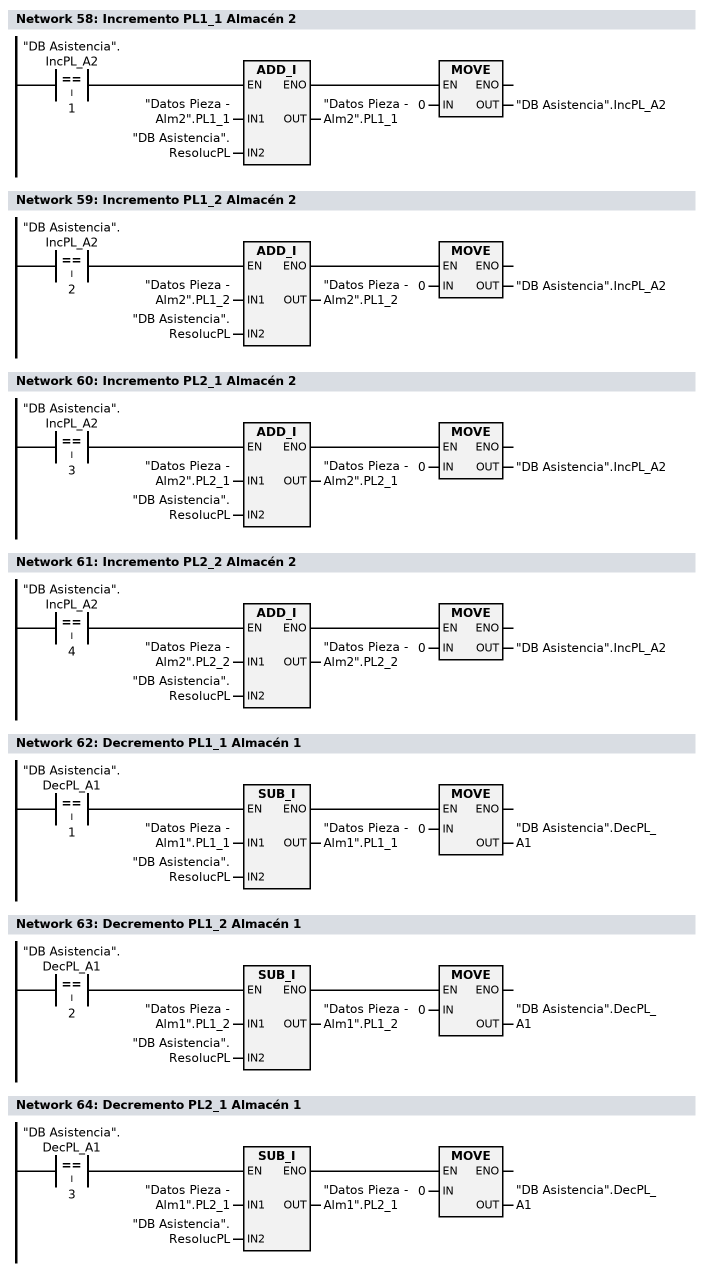
NETWORK
TITLE = Incremento PL1_1 Almacén 2
      A(;
      A(;
      L     "DB Asistencia".IncPL_A2;
      L     1;
      ==I;
      );
      JNB   _03d;
      L     "Datos Pieza - Alm2".PL1_1;
      L     "DB Asistencia".ResolucPL;
      +I;
      T     "Datos Pieza - Alm2".PL1_1;
      AN    OV;
      SAVE;
      CLR;
_03d: A     BR;
      );
      JNB   _03e;
      L     0;
      T     "DB Asistencia".IncPL_A2;
_03e: NOP   0;
NETWORK
TITLE = Incremento PL1_2 Almacén 2
      A(;
      A(;
      L     "DB Asistencia".IncPL_A2;
      L     2;
      ==I;
      );
      JNB   _03f;
      L     "Datos Pieza - Alm2".PL1_2;
      L     "DB Asistencia".ResolucPL;
      +I;
      T     "Datos Pieza - Alm2".PL1_2;
      AN    OV;
      SAVE;
      CLR;
_03f: A     BR;
      );
      JNB   _040;
      L     0;
      T     "DB Asistencia".IncPL_A2;
_040: NOP   0;
NETWORK
TITLE = Incremento PL2_1 Almacén 2
      A(;
      A(;
      L     "DB Asistencia".IncPL_A2;
      L     3;
      ==I;
      );
      JNB   _041;
      L     "Datos Pieza - Alm2".PL2_1;
      L     "DB Asistencia".ResolucPL;
      +I;
      T     "Datos Pieza - Alm2".PL2_1;
      AN    OV;
      SAVE;
      CLR;
_041: A     BR;
      );
      JNB   _042;
      L     0;
      T     "DB Asistencia".IncPL_A2;
_042: NOP   0;
NETWORK
TITLE = Incremento PL2_2 Almacén 2
      A(;
      A(;
      L     "DB Asistencia".IncPL_A2;
      L     4;
      ==I;
      );
      JNB   _043;
      L     "Datos Pieza - Alm2".PL2_2;
      L     "DB Asistencia".ResolucPL;
      +I;
      T     "Datos Pieza - Alm2".PL2_2;
      AN    OV;
      SAVE;
      CLR;
_043: A     BR;
      );
      JNB   _044;
      L     0;
      T     "DB Asistencia".IncPL_A2;
_044: NOP   0;
NETWORK
TITLE = Decremento PL1_1 Almacén 1
      A(;
      A(;
      L     "DB Asistencia".DecPL_A1;
      L     1;
      ==I;
      );
      JNB   _045;
      L     "Datos Pieza - Alm1".PL1_1;
      L     "DB Asistencia".ResolucPL;
      -I;
      T     "Datos Pieza - Alm1".PL1_1;
      AN    OV;
      SAVE;
      CLR;
_045: A     BR;
      );
      JNB   _046;
      L     0;
      T     "DB Asistencia".DecPL_A1;
_046: NOP   0;
NETWORK
TITLE = Decremento PL1_2 Almacén 1
      A(;
      A(;
      L     "DB Asistencia".DecPL_A1;
      L     2;
      ==I;
      );
      JNB   _047;
      L     "Datos Pieza - Alm1".PL1_2;
      L     "DB Asistencia".ResolucPL;
      -I;
      T     "Datos Pieza - Alm1".PL1_2;
      AN    OV;
      SAVE;
      CLR;
_047: A     BR;
      );
      JNB   _048;
      L     0;
      T     "DB Asistencia".DecPL_A1;
_048: NOP   0;
NETWORK
TITLE = Decremento PL2_1 Almacén 1
      A(;
      A(;
      L     "DB Asistencia".DecPL_A1;
      L     3;
      ==I;
      );
      JNB   _049;
      L     "Datos Pieza - Alm1".PL2_1;
      L     "DB Asistencia".ResolucPL;
      -I;
      T     "Datos Pieza - Alm1".PL2_1;
      AN    OV;
      SAVE;
      CLR;
_049: A     BR;
      );
      JNB   _04a;
      L     0;
      T     "DB Asistencia".DecPL_A1;
_04a: NOP   0;
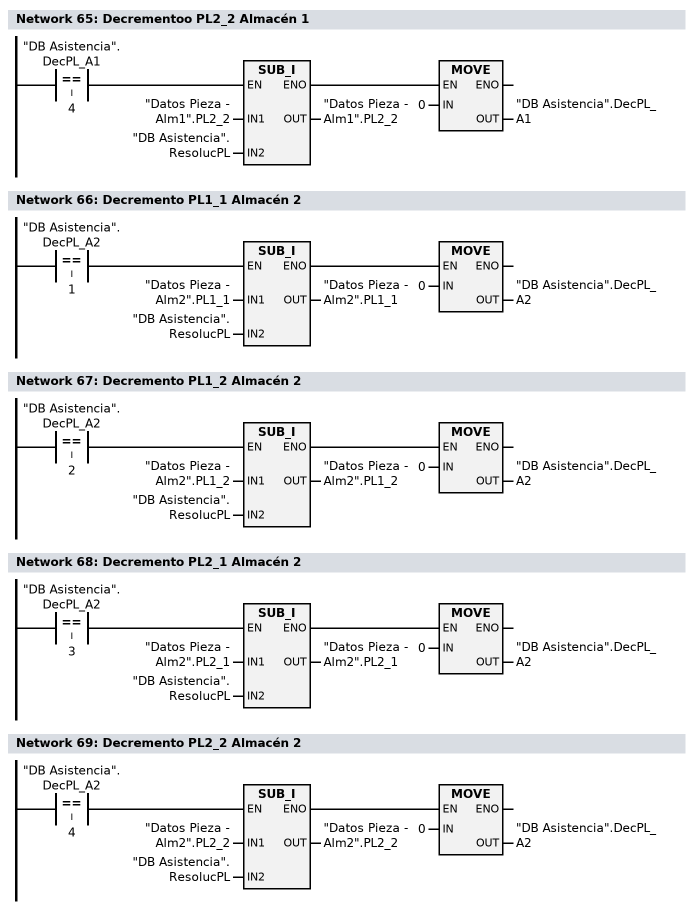
NETWORK
TITLE = Decrementoo PL2_2 Almacén 1
      A(;
      A(;
      L     "DB Asistencia".DecPL_A1;
      L     4;
      ==I;
      );
      JNB   _04b;
      L     "Datos Pieza - Alm1".PL2_2;
      L     "DB Asistencia".ResolucPL;
      -I;
      T     "Datos Pieza - Alm1".PL2_2;
      AN    OV;
      SAVE;
      CLR;
_04b: A     BR;
      );
      JNB   _04c;
      L     0;
      T     "DB Asistencia".DecPL_A1;
_04c: NOP   0;
NETWORK
TITLE = Decremento PL1_1 Almacén 2
      A(;
      A(;
      L     "DB Asistencia".DecPL_A2;
      L     1;
      ==I;
      );
      JNB   _04d;
      L     "Datos Pieza - Alm2".PL1_1;
      L     "DB Asistencia".ResolucPL;
      -I;
      T     "Datos Pieza - Alm2".PL1_1;
      AN    OV;
      SAVE;
      CLR;
_04d: A     BR;
      );
      JNB   _04e;
      L     0;
      T     "DB Asistencia".DecPL_A2;
_04e: NOP   0;
NETWORK
TITLE = Decremento PL1_2 Almacén 2
      A(;
      A(;
      L     "DB Asistencia".DecPL_A2;
      L     2;
      ==I;
      );
      JNB   _04f;
      L     "Datos Pieza - Alm2".PL1_2;
      L     "DB Asistencia".ResolucPL;
      -I;
      T     "Datos Pieza - Alm2".PL1_2;
      AN    OV;
      SAVE;
      CLR;
_04f: A     BR;
      );
      JNB   _050;
      L     0;
      T     "DB Asistencia".DecPL_A2;
_050: NOP   0;
NETWORK
TITLE = Decremento PL2_1 Almacén 2
      A(;
      A(;
      L     "DB Asistencia".DecPL_A2;
      L     3;
      ==I;
      );
      JNB   _051;
      L     "Datos Pieza - Alm2".PL2_1;
      L     "DB Asistencia".ResolucPL;
      -I;
      T     "Datos Pieza - Alm2".PL2_1;
      AN    OV;
      SAVE;
      CLR;
_051: A     BR;
      );
      JNB   _052;
      L     0;
      T     "DB Asistencia".DecPL_A2;
_052: NOP   0;
NETWORK
TITLE = Decremento PL2_2 Almacén 2
      A(;
      A(;
      L     "DB Asistencia".DecPL_A2;
      L     4;
      ==I;
      );
      JNB   _053;
      L     "Datos Pieza - Alm2".PL2_2;
      L     "DB Asistencia".ResolucPL;
      -I;
      T     "Datos Pieza - Alm2".PL2_2;
      AN    OV;
      SAVE;
      CLR;
_053: A     BR;
      );
      JNB   _054;
      L     0;
      T     "DB Asistencia".DecPL_A2;
_054: NOP   0;
END_FUNCTION

FUNCTION "Control de Plegadora" : VOID	// FC 9
TITLE = Control de Plegadora
AUTHOR : EMR
NAME : eProC
VERSION : 0.1
VAR_TEMP
  AUX_POS_RECEPCION : DINT ;
  AUX_POS_ALINEACION : DINT ;
  AUX_POS_PL1 : DINT ;
  AUX_POS_PL2 : DINT ;
  AUX_POS_ENTREGA : DINT ;
  AUX_SALIDA : DINT ;
  AUX_CHAPA_COMPLETA : DINT ;
  AUX_ESPERA : DINT ;
  PL1_A : DINT ;
  PL1_B : DINT ;
  PL1_C : DINT ;
  PL1_D : DINT ;
  PL1_1 : DINT ;
  PL1_2 : DINT ;
  AUX_ENCODER : REAL ;
  AUX_ENCODER2 : DINT ;
  AUX_REAL : REAL ;
  AUX_REAL2 : REAL ;
  AUX_REAL3 : REAL ;
  PL2_1 : DINT ;
  PL2_2 : DINT ;
  POS_PINZA_SEGURA1 : DINT ;
  POS_PINZA_SEGURA2 : DINT ;
  AUX_DINT : DINT ;
  AUX_POS_RECEP : BOOL ;	//Plegadores en Posición Recepción
  AUX_POS_ALIN : BOOL ;	//Plegadores en Posición Alineación
  AUX_POS_ENT : BOOL ;	//Plegadores en Posición Entrega
  AUX_POS_ESP : BOOL ;	//Plegadores en Posición Espera
  AUX_POS_26 : BOOL ;
  AUX_POS_25 : BOOL ;
  AUX_POS_PLEG2 : BOOL ;	//Plegadores en Posición Plegado 2
  AUX_POS_24 : BOOL ;
  AUX_POS_22 : BOOL ;
  AUX_POS_PLEG1 : BOOL ;	//Plegadores en Posición Plegado 1
  AUX_POS_23 : BOOL ;
  AUX_POS_21 : BOOL ;
END_VAR
BEGIN
NETWORK
TITLE = ------------- HABILITACIÓN SERVOS -----------------
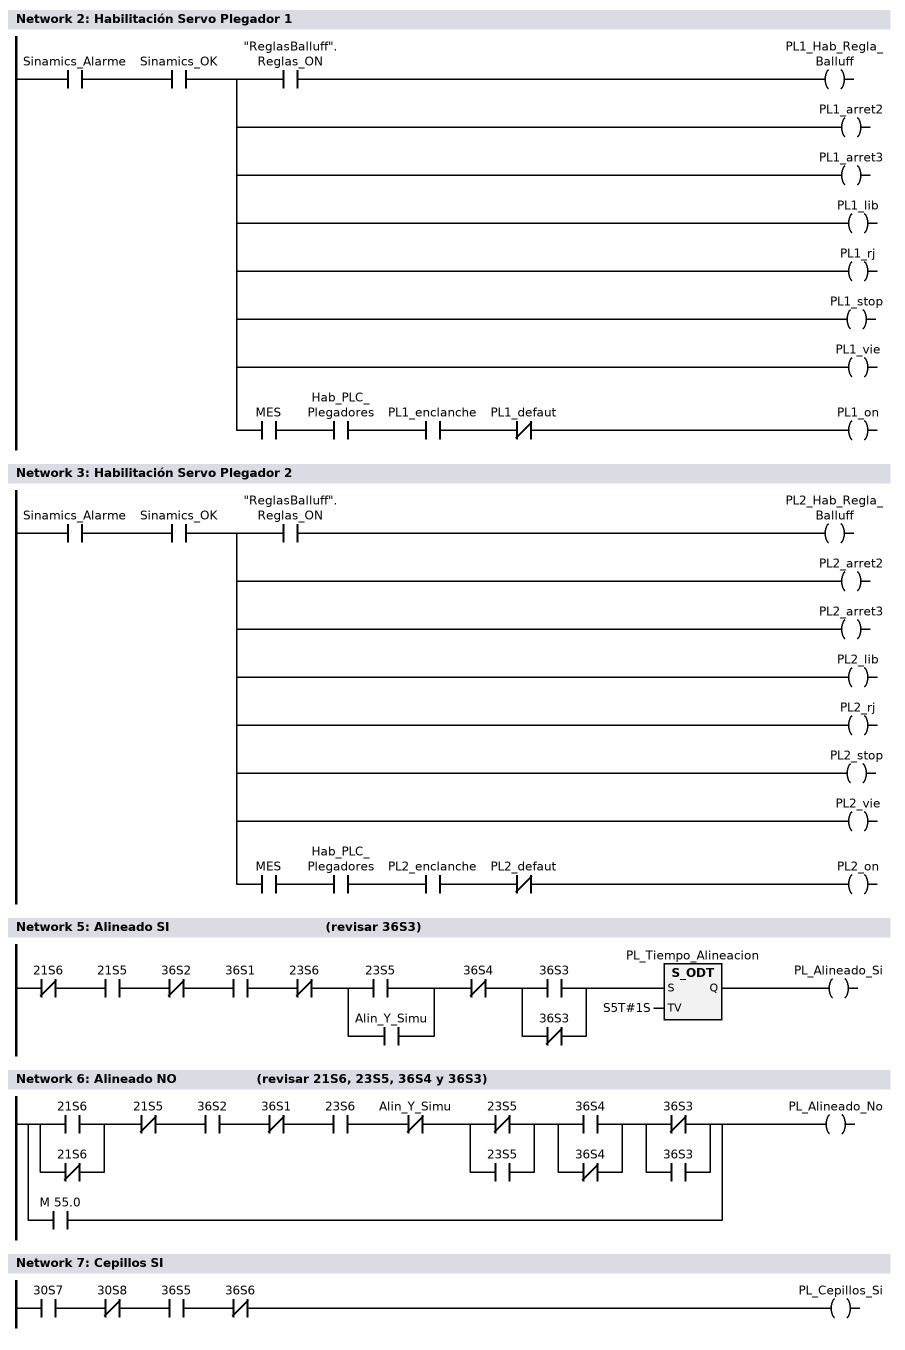
NETWORK
TITLE = Habilitación Servo Plegador 1
      A     "Sinamics_Alarme";
      A     "Sinamics_OK";
      =     L 98.0;
      A     L 98.0;
      A     "ReglasBalluff".Reglas_ON;
      =     "PL1_Hab_Regla_Balluff";
      A     L 98.0;
      BLD   102;
      =     "PL1_arret2";
      A     L 98.0;
      BLD   102;
      =     "PL1_arret3";
      A     L 98.0;
      BLD   102;
      =     "PL1_lib";
      A     L 98.0;
      BLD   102;
      =     "PL1_rj";
      A     L 98.0;
      BLD   102;
      =     "PL1_stop";
      A     L 98.0;
      BLD   102;
      =     "PL1_vie";
      A     L 98.0;
      A     "MES";
      A     "Hab_PLC_Plegadores";
      A     "PL1_enclanche";
      AN    "PL1_defaut";
      =     "PL1_on";
NETWORK
TITLE = Habilitación Servo Plegador 2
      A     "Sinamics_Alarme";
      A     "Sinamics_OK";
      =     L 98.0;
      A     L 98.0;
      A     "ReglasBalluff".Reglas_ON;
      =     "PL2_Hab_Regla_Balluff";
      A     L 98.0;
      BLD   102;
      =     "PL2_arret2";
      A     L 98.0;
      BLD   102;
      =     "PL2_arret3";
      A     L 98.0;
      BLD   102;
      =     "PL2_lib";
      A     L 98.0;
      BLD   102;
      =     "PL2_rj";
      A     L 98.0;
      BLD   102;
      =     "PL2_stop";
      A     L 98.0;
      BLD   102;
      =     "PL2_vie";
      A     L 98.0;
      A     "MES";
      A     "Hab_PLC_Plegadores";
      A     "PL2_enclanche";
      AN    "PL2_defaut";
      =     "PL2_on";
NETWORK
TITLE = ------------- RESUMEN DE SENSORES -----------------
NETWORK
TITLE = Alineado SI                                       (revisar 36S3)
      AN    "21S6";
      A     "21S5";
      AN    "36S2";
      A     "36S1";
      AN    "23S6";
      A(;
      O     "23S5";
      O     "Alin_Y_Simu";
      );
      AN    "36S4";
      A(;
      O     "36S3";
      ON    "36S3";
      );
      L     S5T#1S;
      SD    "PL_Tiempo_Alineacion";
      NOP   0;
      NOP   0;
      NOP   0;
      A     "PL_Tiempo_Alineacion";
      =     "PL_Alineado_Si";
NETWORK
TITLE = Alineado NO                    (revisar 21S6, 23S5, 36S4 y 36S3)
      A(;
      O     "21S6";
      ON    "21S6";
      );
      AN    "21S5";
      A     "36S2";
      AN    "36S1";
      A     "23S6";
      AN    "Alin_Y_Simu";
      A(;
      ON    "23S5";
      O     "23S5";
      );
      A(;
      O     "36S4";
      ON    "36S4";
      );
      A(;
      ON    "36S3";
      O     "36S3";
      );
      O     M 55.0;
      =     "PL_Alineado_No";
NETWORK
TITLE = Cepillos SI
      A     "30S7";
      AN    "30S8";
      A     "36S5";
      AN    "36S6";
      =     "PL_Cepillos_Si";
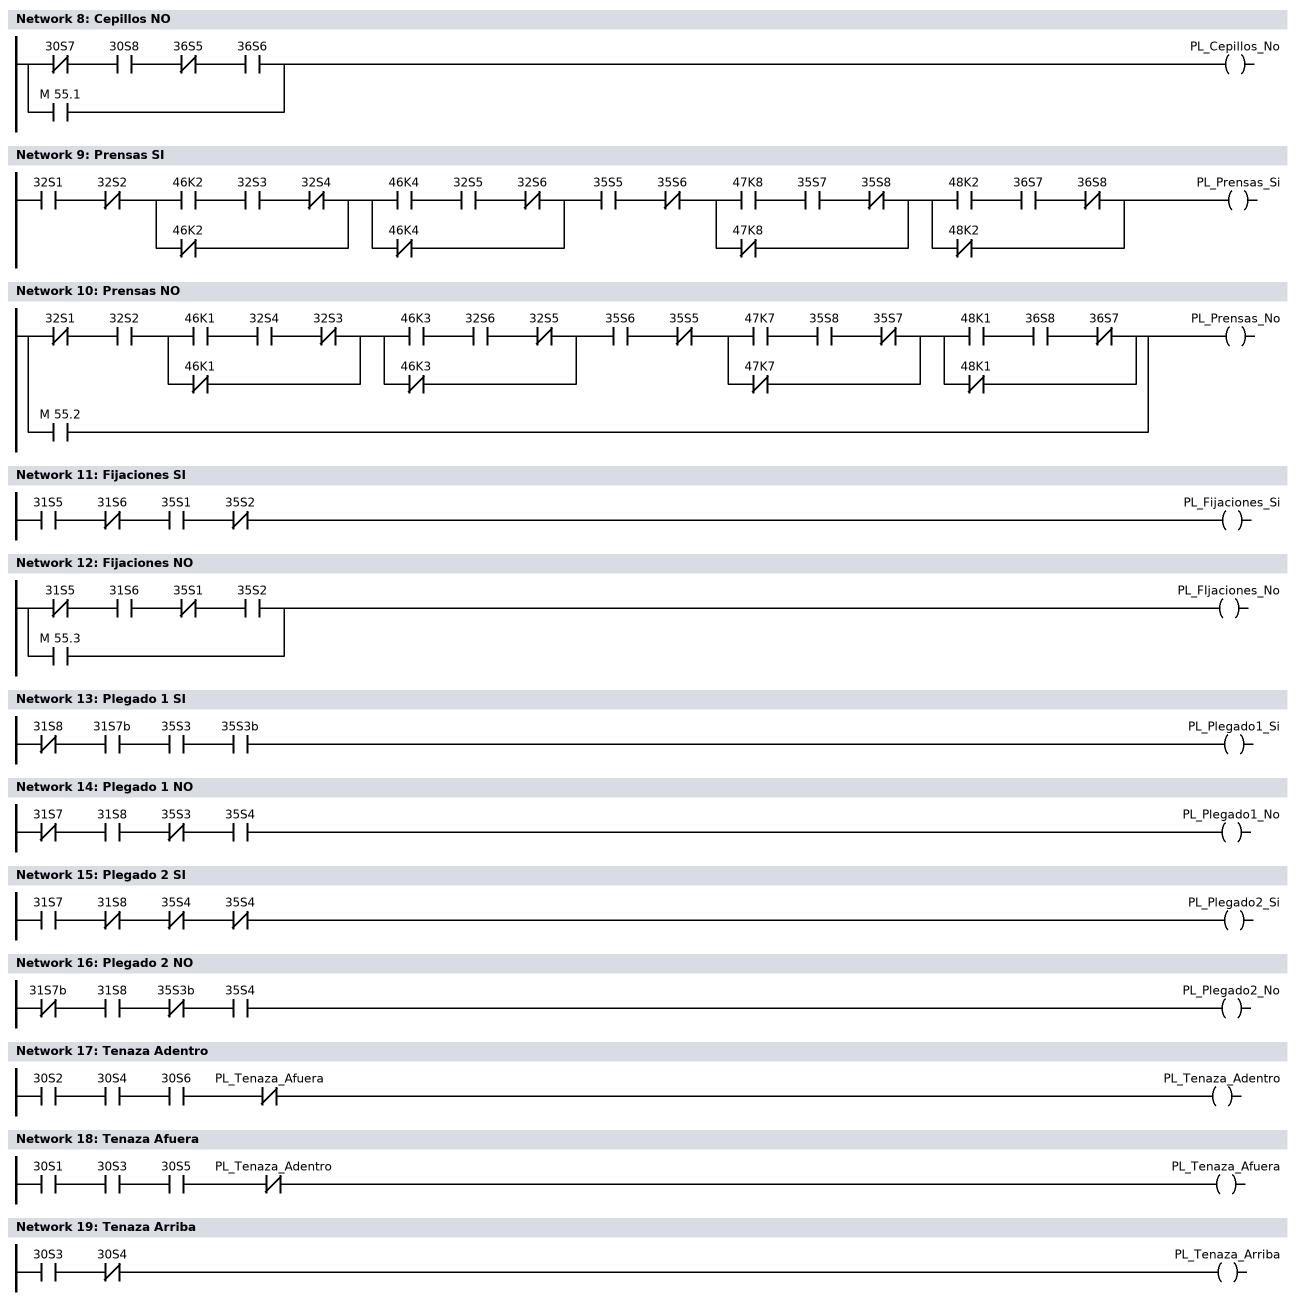
NETWORK
TITLE = Cepillos NO
      AN    "30S7";
      A     "30S8";
      AN    "36S5";
      A     "36S6";
      O     M 55.1;
      =     "PL_Cepillos_No";
NETWORK
TITLE = Prensas SI
      A     "32S1";
      AN    "32S2";
      A(;
      A     "46K2";
      A     "32S3";
      AN    "32S4";
      ON    "46K2";
      );
      A(;
      A     "46K4";
      A     "32S5";
      AN    "32S6";
      ON    "46K4";
      );
      A     "35S5";
      AN    "35S6";
      A(;
      A     "47K8";
      A     "35S7";
      AN    "35S8";
      ON    "47K8";
      );
      A(;
      A     "48K2";
      A     "36S7";
      AN    "36S8";
      ON    "48K2";
      );
      =     "PL_Prensas_Si";
NETWORK
TITLE = Prensas NO
      AN    "32S1";
      A     "32S2";
      A(;
      A     "46K1";
      A     "32S4";
      AN    "32S3";
      ON    "46K1";
      );
      A(;
      A     "46K3";
      A     "32S6";
      AN    "32S5";
      ON    "46K3";
      );
      A     "35S6";
      AN    "35S5";
      A(;
      A     "47K7";
      A     "35S8";
      AN    "35S7";
      ON    "47K7";
      );
      A(;
      A     "48K1";
      A     "36S8";
      AN    "36S7";
      ON    "48K1";
      );
      O     M 55.2;
      =     "PL_Prensas_No";
NETWORK
TITLE = Fijaciones SI
      A     "31S5";
      AN    "31S6";
      A     "35S1";
      AN    "35S2";
      =     "PL_Fijaciones_Si";
NETWORK
TITLE = Fijaciones NO
      AN    "31S5";
      A     "31S6";
      AN    "35S1";
      A     "35S2";
      O     M 55.3;
      =     "PL_FIjaciones_No";
NETWORK
TITLE = Plegado 1 SI
      AN    "31S8";
      A     "31S7b";
      A     "35S3";
      A     "35S3b";
      =     "PL_Plegado1_Si";
NETWORK
TITLE = Plegado 1 NO
      AN    "31S7";
      A     "31S8";
      AN    "35S3";
      A     "35S4";
      =     "PL_Plegado1_No";
NETWORK
TITLE = Plegado 2 SI
      A     "31S7";
      AN    "31S8";
      AN    "35S4";
      AN    "35S4";
      =     "PL_Plegado2_Si";
NETWORK
TITLE = Plegado 2 NO
      AN    "31S7b";
      A     "31S8";
      AN    "35S3b";
      A     "35S4";
      =     "PL_Plegado2_No";
NETWORK
TITLE = Tenaza Adentro
      A     "30S2";
      A     "30S4";
      A     "30S6";
      AN    "PL_Tenaza_Afuera";
      =     "PL_Tenaza_Adentro";
NETWORK
TITLE = Tenaza Afuera
      A     "30S1";
      A     "30S3";
      A     "30S5";
      AN    "PL_Tenaza_Adentro";
      =     "PL_Tenaza_Afuera";
NETWORK
TITLE = Tenaza Arriba
      A     "30S3";
      AN    "30S4";
      =     "PL_Tenaza_Arriba";
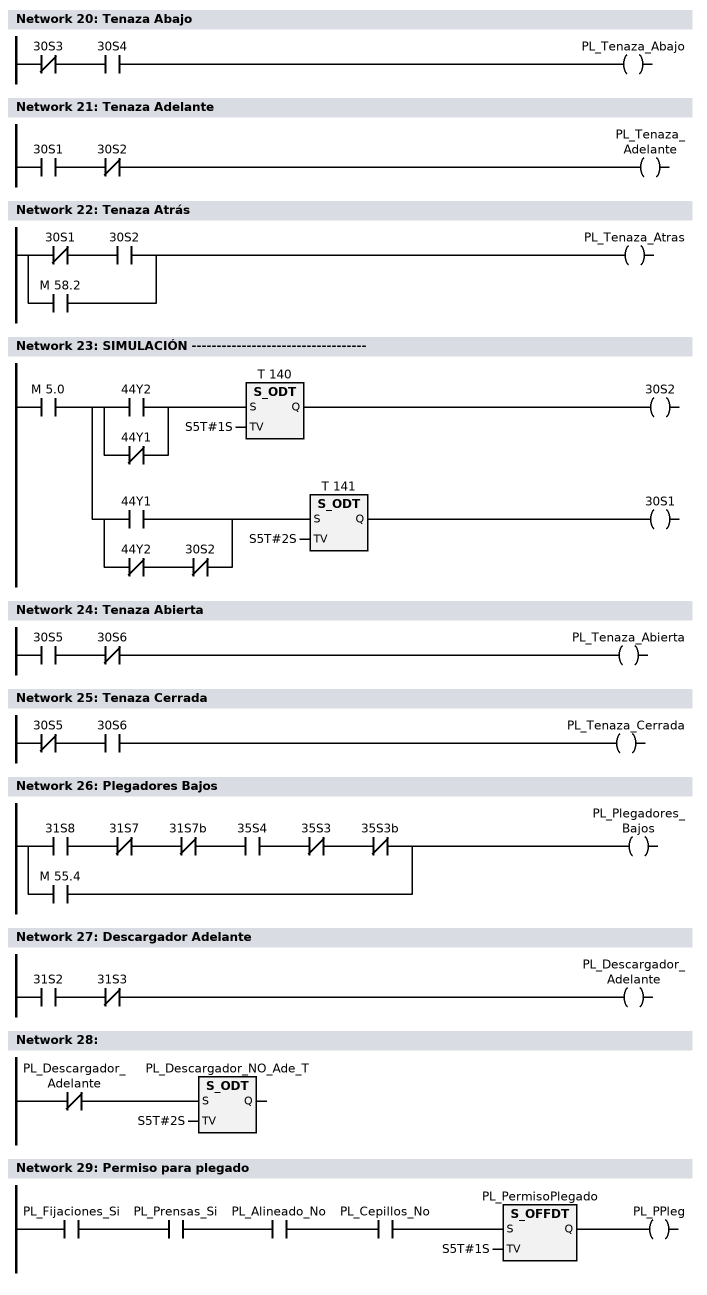
NETWORK
TITLE = Tenaza Abajo
      AN    "30S3";
      A     "30S4";
      =     "PL_Tenaza_Abajo";
NETWORK
TITLE = Tenaza Adelante
      A     "30S1";
      AN    "30S2";
      =     "PL_Tenaza_Adelante";
NETWORK
TITLE = Tenaza Atrás
      AN    "30S1";
      A     "30S2";
      O     M 58.2;
      =     "PL_Tenaza_Atras";
NETWORK
TITLE = SIMULACIÓN -----------------------------------
      A     M 5.0;
      =     L 98.0;
      A     L 98.0;
      A(;
      O     "44Y2";
      ON    "44Y1";
      );
      L     S5T#1S;
      SD    T 140;
      NOP   0;
      NOP   0;
      NOP   0;
      A     T 140;
      =     "30S2";
      A     L 98.0;
      A(;
      O     "44Y1";
      O;
      AN    "44Y2";
      AN    "30S2";
      );
      L     S5T#2S;
      SD    T 141;
      NOP   0;
      NOP   0;
      NOP   0;
      A     T 141;
      =     "30S1";
NETWORK
TITLE = Tenaza Abierta
      A     "30S5";
      AN    "30S6";
      =     "PL_Tenaza_Abierta";
NETWORK
TITLE = Tenaza Cerrada
      AN    "30S5";
      A     "30S6";
      =     "PL_Tenaza_Cerrada";
NETWORK
TITLE = Plegadores Bajos
      A     "31S8";
      AN    "31S7";
      AN    "31S7b";
      A     "35S4";
      AN    "35S3";
      AN    "35S3b";
      O     M 55.4;
      =     "PL_Plegadores_Bajos";
NETWORK
TITLE = Descargador Adelante
      A     "31S2";
      AN    "31S3";
      =     "PL_Descargador_Adelante";
NETWORK
TITLE =
      AN    "PL_Descargador_Adelante";
      L     S5T#2S;
      SD    "PL_Descargador_NO_Ade_T";
      NOP   0;
      NOP   0;
      NOP   0;
      NOP   0;
NETWORK
TITLE = Permiso para plegado
      A     "PL_Fijaciones_Si";
      A     "PL_Prensas_Si";
      A     "PL_Alineado_No";
      A     "PL_Cepillos_No";
      L     S5T#1S;
      SF    "PL_PermisoPlegado";
      NOP   0;
      NOP   0;
      NOP   0;
      A     "PL_PermisoPlegado";
      =     "PL_PPleg";
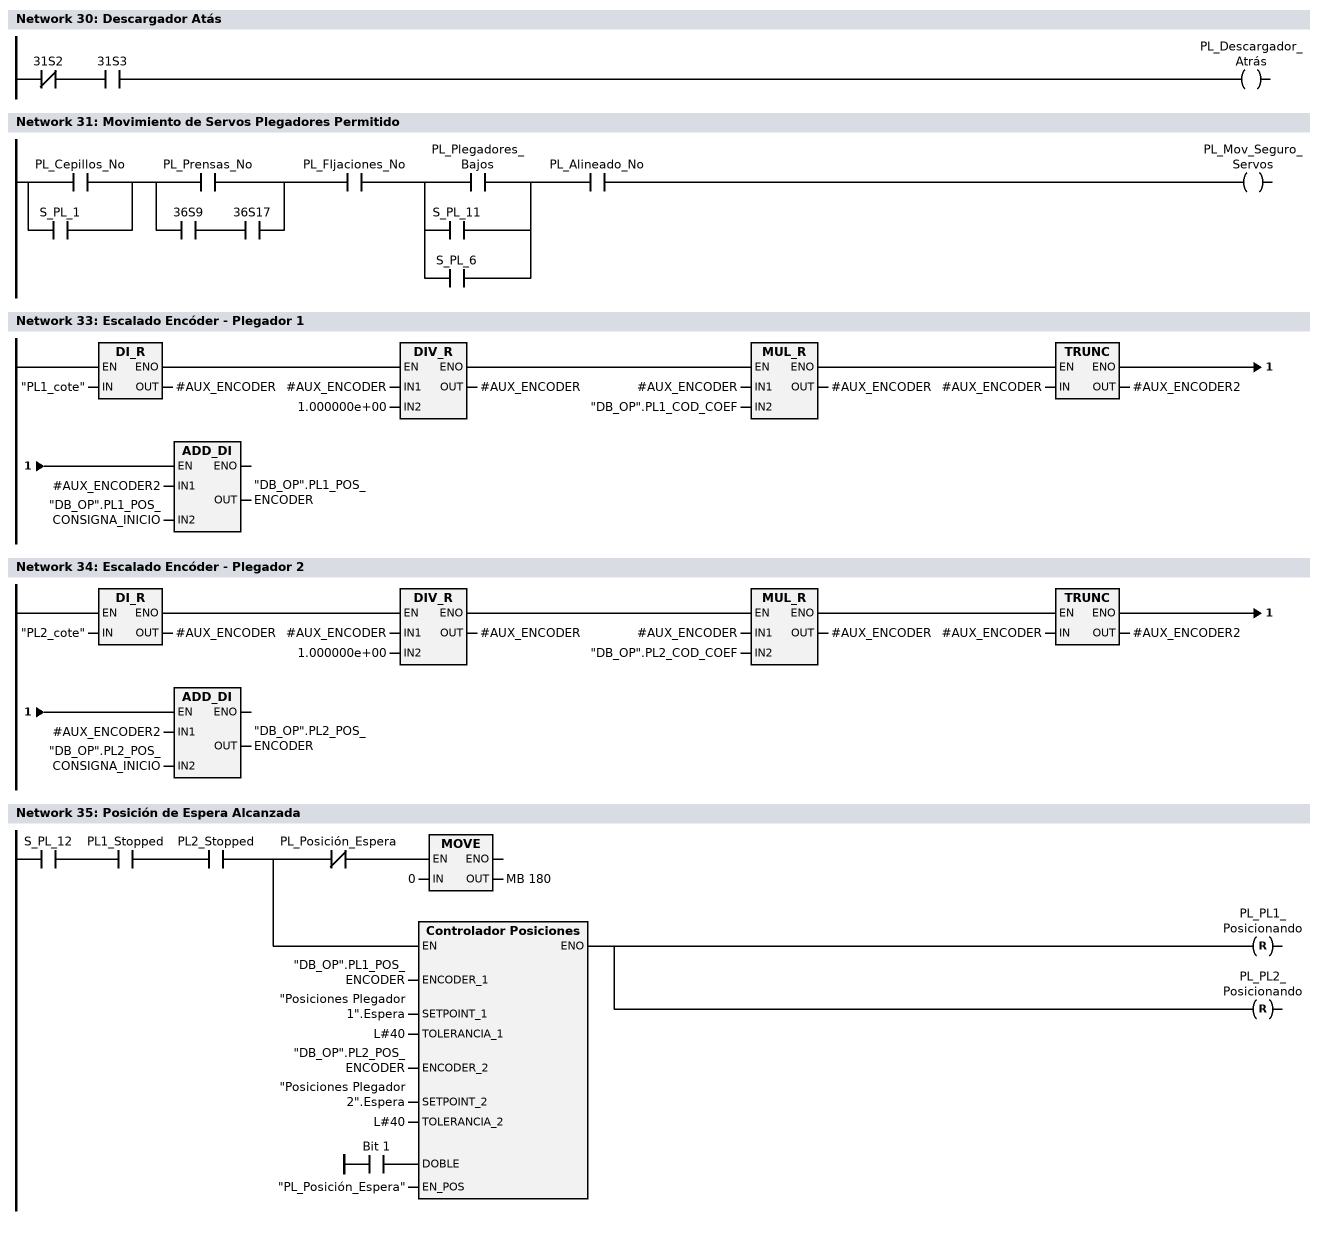
NETWORK
TITLE = Descargador Atás
      AN    "31S2";
      A     "31S3";
      =     "PL_Descargador_Atrás";
NETWORK
TITLE = Movimiento de Servos Plegadores Permitido
      A(;
      O     "PL_Cepillos_No";
      O     "S_PL_1";
      );
      A(;
      O     "PL_Prensas_No";
      O;
      A     "36S9";
      A     "36S17";
      );
      A     "PL_FIjaciones_No";
      A(;
      O     "PL_Plegadores_Bajos";
      O     "S_PL_11";
      O     "S_PL_6";
      );
      A     "PL_Alineado_No";
      =     "PL_Mov_Seguro_Servos";
NETWORK
TITLE = ------------ ESCALADO DE ENCODERS -------------
NETWORK
TITLE = Escalado Encóder - Plegador 1
      A(;
      A(;
      A(;
      A(;
      L     "PL1_cote";
      DTR;
      T     #AUX_ENCODER;
      SET;
      SAVE;
      CLR;
      A     BR;
      );
      JNB   _001;
      L     #AUX_ENCODER;
      L     1.000000e+00;
      /R;
      T     #AUX_ENCODER;
      AN    OV;
      SAVE;
      CLR;
_001: A     BR;
      );
      JNB   _002;
      L     #AUX_ENCODER;
      L     "DB_OP".PL1_COD_COEF;
      *R;
      T     #AUX_ENCODER;
      AN    OV;
      SAVE;
      CLR;
_002: A     BR;
      );
      JNB   _003;
      L     #AUX_ENCODER;
      TRUNC;
      T     #AUX_ENCODER2;
      AN    OV;
      SAVE;
      CLR;
_003: A     BR;
      );
      JNB   _004;
      L     #AUX_ENCODER2;
      L     "DB_OP".PL1_POS_CONSIGNA_INICIO;
      +D;
      T     "DB_OP".PL1_POS_ENCODER;
_004: NOP   0;
NETWORK
TITLE = Escalado Encóder - Plegador 2
      A(;
      A(;
      A(;
      A(;
      L     "PL2_cote";
      DTR;
      T     #AUX_ENCODER;
      SET;
      SAVE;
      CLR;
      A     BR;
      );
      JNB   _005;
      L     #AUX_ENCODER;
      L     1.000000e+00;
      /R;
      T     #AUX_ENCODER;
      AN    OV;
      SAVE;
      CLR;
_005: A     BR;
      );
      JNB   _006;
      L     #AUX_ENCODER;
      L     "DB_OP".PL2_COD_COEF;
      *R;
      T     #AUX_ENCODER;
      AN    OV;
      SAVE;
      CLR;
_006: A     BR;
      );
      JNB   _007;
      L     #AUX_ENCODER;
      TRUNC;
      T     #AUX_ENCODER2;
      AN    OV;
      SAVE;
      CLR;
_007: A     BR;
      );
      JNB   _008;
      L     #AUX_ENCODER2;
      L     "DB_OP".PL2_POS_CONSIGNA_INICIO;
      +D;
      T     "DB_OP".PL2_POS_ENCODER;
_008: NOP   0;
NETWORK
TITLE = Posición de Espera Alcanzada
      A     "S_PL_12";
      A     "PL1_Stopped";
      A     "PL2_Stopped";
      =     L 98.0;
      A     L 98.0;
      AN    "PL_Posición_Espera";
      JNB   _009;
      L     0;
      T     MB 180;
_009: NOP   0;
      A     "Bit 1";
      =     L 98.1;
      BLD   103;
      A     L 98.0;
      JNB   _00a;
      CALL  "Controlador Posiciones" (
           ENCODER_1                := "DB_OP".PL1_POS_ENCODER,
           SETPOINT_1               := "Posiciones Plegador 1".Espera,
           TOLERANCIA_1             := L#40,
           ENCODER_2                := "DB_OP".PL2_POS_ENCODER,
           SETPOINT_2               := "Posiciones Plegador 2".Espera,
           TOLERANCIA_2             := L#40,
           DOBLE                    := L 98.1,
           EN_POS                   := "PL_Posición_Espera");
_00a: A     BR;
      R     "PL_PL1_Posicionando";
      R     "PL_PL2_Posicionando";
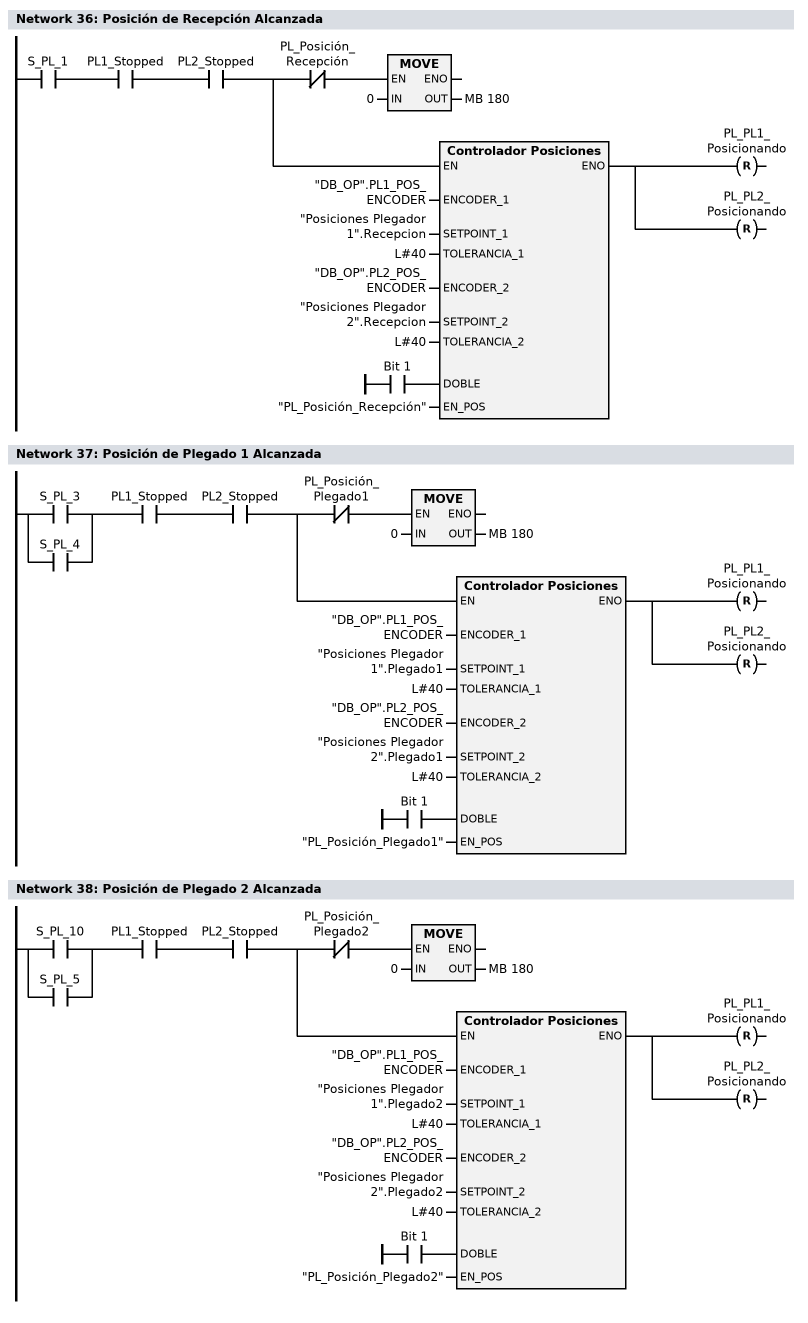
NETWORK
TITLE = Posición de Recepción Alcanzada
      A     "S_PL_1";
      A     "PL1_Stopped";
      A     "PL2_Stopped";
      =     L 98.0;
      A     L 98.0;
      AN    "PL_Posición_Recepción";
      JNB   _00b;
      L     0;
      T     MB 180;
_00b: NOP   0;
      A     "Bit 1";
      =     L 98.1;
      BLD   103;
      A     L 98.0;
      JNB   _00c;
      CALL  "Controlador Posiciones" (
           ENCODER_1                := "DB_OP".PL1_POS_ENCODER,
           SETPOINT_1               := "Posiciones Plegador 1".Recepcion,
           TOLERANCIA_1             := L#40,
           ENCODER_2                := "DB_OP".PL2_POS_ENCODER,
           SETPOINT_2               := "Posiciones Plegador 2".Recepcion,
           TOLERANCIA_2             := L#40,
           DOBLE                    := L 98.1,
           EN_POS                   := "PL_Posición_Recepción");
_00c: A     BR;
      R     "PL_PL1_Posicionando";
      R     "PL_PL2_Posicionando";
NETWORK
TITLE = Posición de Plegado 1 Alcanzada
      A(;
      O     "S_PL_3";
      O     "S_PL_4";
      );
      A     "PL1_Stopped";
      A     "PL2_Stopped";
      =     L 98.0;
      A     L 98.0;
      AN    "PL_Posición_Plegado1";
      JNB   _00d;
      L     0;
      T     MB 180;
_00d: NOP   0;
      A     "Bit 1";
      =     L 98.1;
      BLD   103;
      A     L 98.0;
      JNB   _00e;
      CALL  "Controlador Posiciones" (
           ENCODER_1                := "DB_OP".PL1_POS_ENCODER,
           SETPOINT_1               := "Posiciones Plegador 1".Plegado1,
           TOLERANCIA_1             := L#40,
           ENCODER_2                := "DB_OP".PL2_POS_ENCODER,
           SETPOINT_2               := "Posiciones Plegador 2".Plegado1,
           TOLERANCIA_2             := L#40,
           DOBLE                    := L 98.1,
           EN_POS                   := "PL_Posición_Plegado1");
_00e: A     BR;
      R     "PL_PL1_Posicionando";
      R     "PL_PL2_Posicionando";
NETWORK
TITLE = Posición de Plegado 2 Alcanzada
      A(;
      O     "S_PL_10";
      O     "S_PL_5";
      );
      A     "PL1_Stopped";
      A     "PL2_Stopped";
      =     L 98.0;
      A     L 98.0;
      AN    "PL_Posición_Plegado2";
      JNB   _00f;
      L     0;
      T     MB 180;
_00f: NOP   0;
      A     "Bit 1";
      =     L 98.1;
      BLD   103;
      A     L 98.0;
      JNB   _010;
      CALL  "Controlador Posiciones" (
           ENCODER_1                := "DB_OP".PL1_POS_ENCODER,
           SETPOINT_1               := "Posiciones Plegador 1".Plegado2,
           TOLERANCIA_1             := L#40,
           ENCODER_2                := "DB_OP".PL2_POS_ENCODER,
           SETPOINT_2               := "Posiciones Plegador 2".Plegado2,
           TOLERANCIA_2             := L#40,
           DOBLE                    := L 98.1,
           EN_POS                   := "PL_Posición_Plegado2");
_010: A     BR;
      R     "PL_PL1_Posicionando";
      R     "PL_PL2_Posicionando";
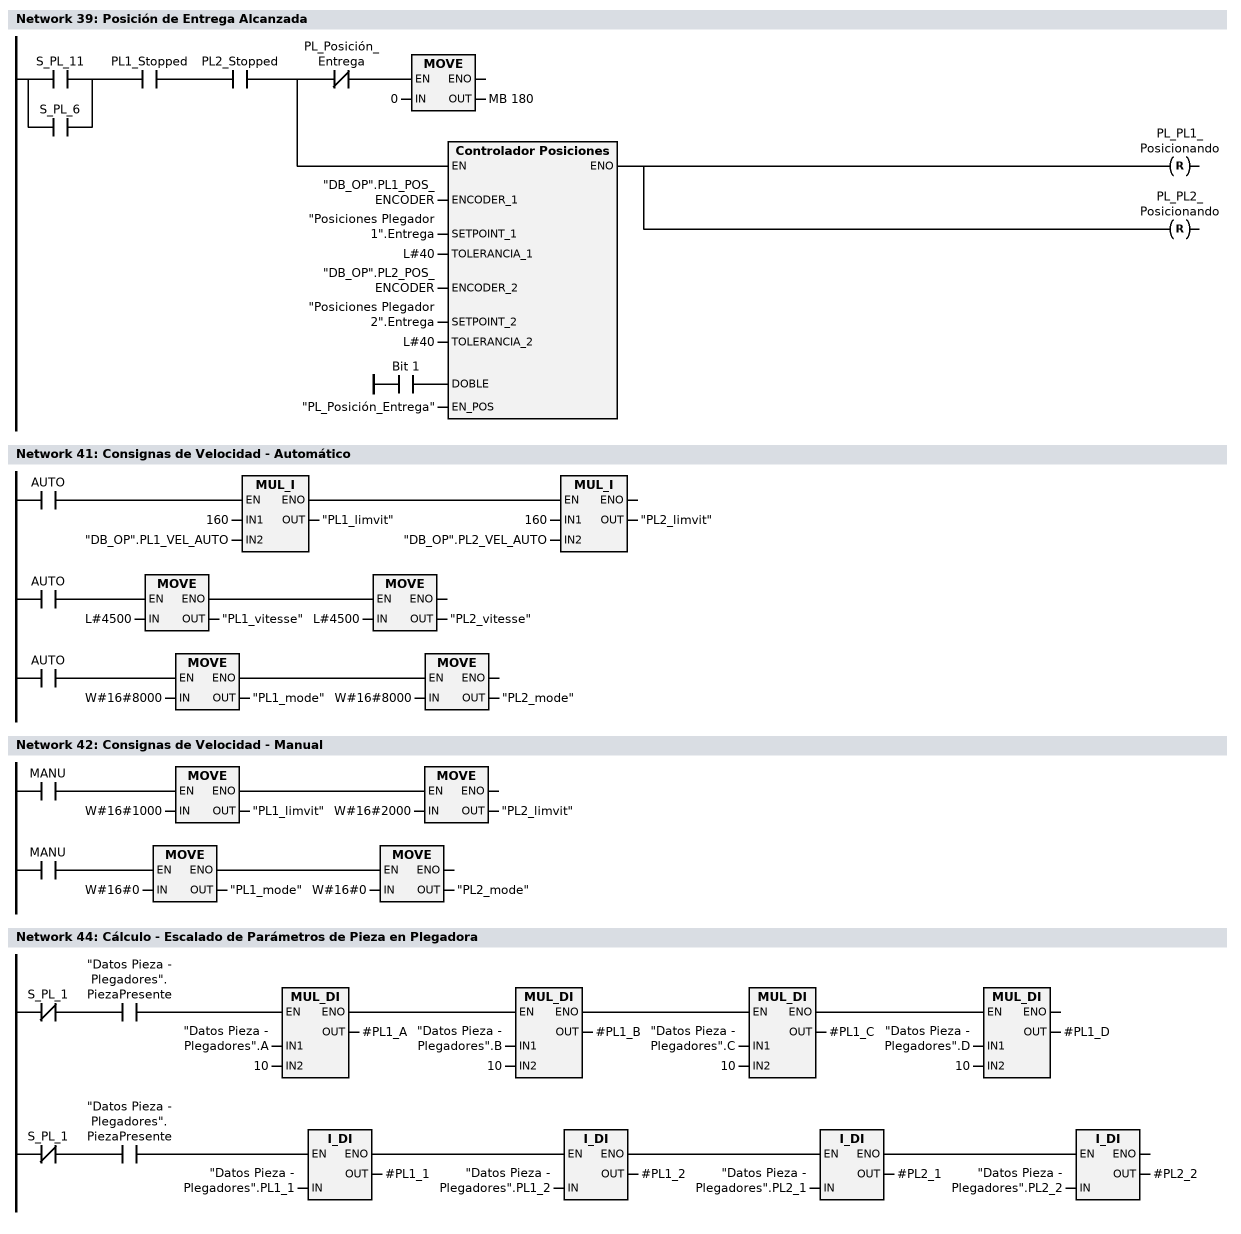
NETWORK
TITLE = Posición de Entrega Alcanzada
      A(;
      O     "S_PL_11";
      O     "S_PL_6";
      );
      A     "PL1_Stopped";
      A     "PL2_Stopped";
      =     L 98.0;
      A     L 98.0;
      AN    "PL_Posición_Entrega";
      JNB   _011;
      L     0;
      T     MB 180;
_011: NOP   0;
      A     "Bit 1";
      =     L 98.1;
      BLD   103;
      A     L 98.0;
      JNB   _012;
      CALL  "Controlador Posiciones" (
           ENCODER_1                := "DB_OP".PL1_POS_ENCODER,
           SETPOINT_1               := "Posiciones Plegador 1".Entrega,
           TOLERANCIA_1             := L#40,
           ENCODER_2                := "DB_OP".PL2_POS_ENCODER,
           SETPOINT_2               := "Posiciones Plegador 2".Entrega,
           TOLERANCIA_2             := L#40,
           DOBLE                    := L 98.1,
           EN_POS                   := "PL_Posición_Entrega");
_012: A     BR;
      R     "PL_PL1_Posicionando";
      R     "PL_PL2_Posicionando";
NETWORK
TITLE = ------------ CONSIGNAS DE VELOCIDAD -----------
NETWORK
TITLE = Consignas de Velocidad - Automático
      A     "AUTO";
      =     L 98.0;
      A(;
      A     L 98.0;
      JNB   _013;
      L     160;
      L     "DB_OP".PL1_VEL_AUTO;
      *I;
      T     "PL1_limvit";
      AN    OV;
      SAVE;
      CLR;
_013: A     BR;
      );
      JNB   _014;
      L     160;
      L     "DB_OP".PL2_VEL_AUTO;
      *I;
      T     "PL2_limvit";
_014: NOP   0;
      A(;
      A     L 98.0;
      JNB   _015;
      L     L#4500;
      T     "PL1_vitesse";
      SET;
      SAVE;
      CLR;
_015: A     BR;
      );
      JNB   _016;
      L     L#4500;
      T     "PL2_vitesse";
_016: NOP   0;
      A(;
      A     L 98.0;
      JNB   _017;
      L     W#16#8000;
      T     "PL1_mode";
      SET;
      SAVE;
      CLR;
_017: A     BR;
      );
      JNB   _018;
      L     W#16#8000;
      T     "PL2_mode";
_018: NOP   0;
NETWORK
TITLE = Consignas de Velocidad - Manual
      A     "MANU";
      =     L 98.0;
      A(;
      A     L 98.0;
      JNB   _019;
      L     W#16#1000;
      T     "PL1_limvit";
      SET;
      SAVE;
      CLR;
_019: A     BR;
      );
      JNB   _01a;
      L     W#16#2000;
      T     "PL2_limvit";
_01a: NOP   0;
      A(;
      A     L 98.0;
      JNB   _01b;
      L     W#16#0;
      T     "PL1_mode";
      SET;
      SAVE;
      CLR;
_01b: A     BR;
      );
      JNB   _01c;
      L     W#16#0;
      T     "PL2_mode";
_01c: NOP   0;
NETWORK
TITLE = ------------ CÁLCULO DE REFERENCIAS -----------
NETWORK
TITLE = Cálculo - Escalado de Parámetros de Pieza en Plegadora
      AN    "S_PL_1";
      A     "Datos Pieza - Plegadores".PiezaPresente;
      =     L 98.0;
      A(;
      A(;
      A(;
      A     L 98.0;
      JNB   _01d;
      L     "Datos Pieza - Plegadores".A;
      L     10;
      *D;
      T     #PL1_A;
      AN    OV;
      SAVE;
      CLR;
_01d: A     BR;
      );
      JNB   _01e;
      L     "Datos Pieza - Plegadores".B;
      L     10;
      *D;
      T     #PL1_B;
      AN    OV;
      SAVE;
      CLR;
_01e: A     BR;
      );
      JNB   _01f;
      L     "Datos Pieza - Plegadores".C;
      L     10;
      *D;
      T     #PL1_C;
      AN    OV;
      SAVE;
      CLR;
_01f: A     BR;
      );
      JNB   _020;
      L     "Datos Pieza - Plegadores".D;
      L     10;
      *D;
      T     #PL1_D;
_020: NOP   0;
      A(;
      A(;
      A(;
      A     L 98.0;
      JNB   _021;
      L     "Datos Pieza - Plegadores".PL1_1;
      ITD;
      T     #PL1_1;
      SET;
      SAVE;
      CLR;
_021: A     BR;
      );
      JNB   _022;
      L     "Datos Pieza - Plegadores".PL1_2;
      ITD;
      T     #PL1_2;
      SET;
      SAVE;
      CLR;
_022: A     BR;
      );
      JNB   _023;
      L     "Datos Pieza - Plegadores".PL2_1;
      ITD;
      T     #PL2_1;
      SET;
      SAVE;
      CLR;
_023: A     BR;
      );
      JNB   _024;
      L     "Datos Pieza - Plegadores".PL2_2;
      ITD;
      T     #PL2_2;
_024: NOP   0;
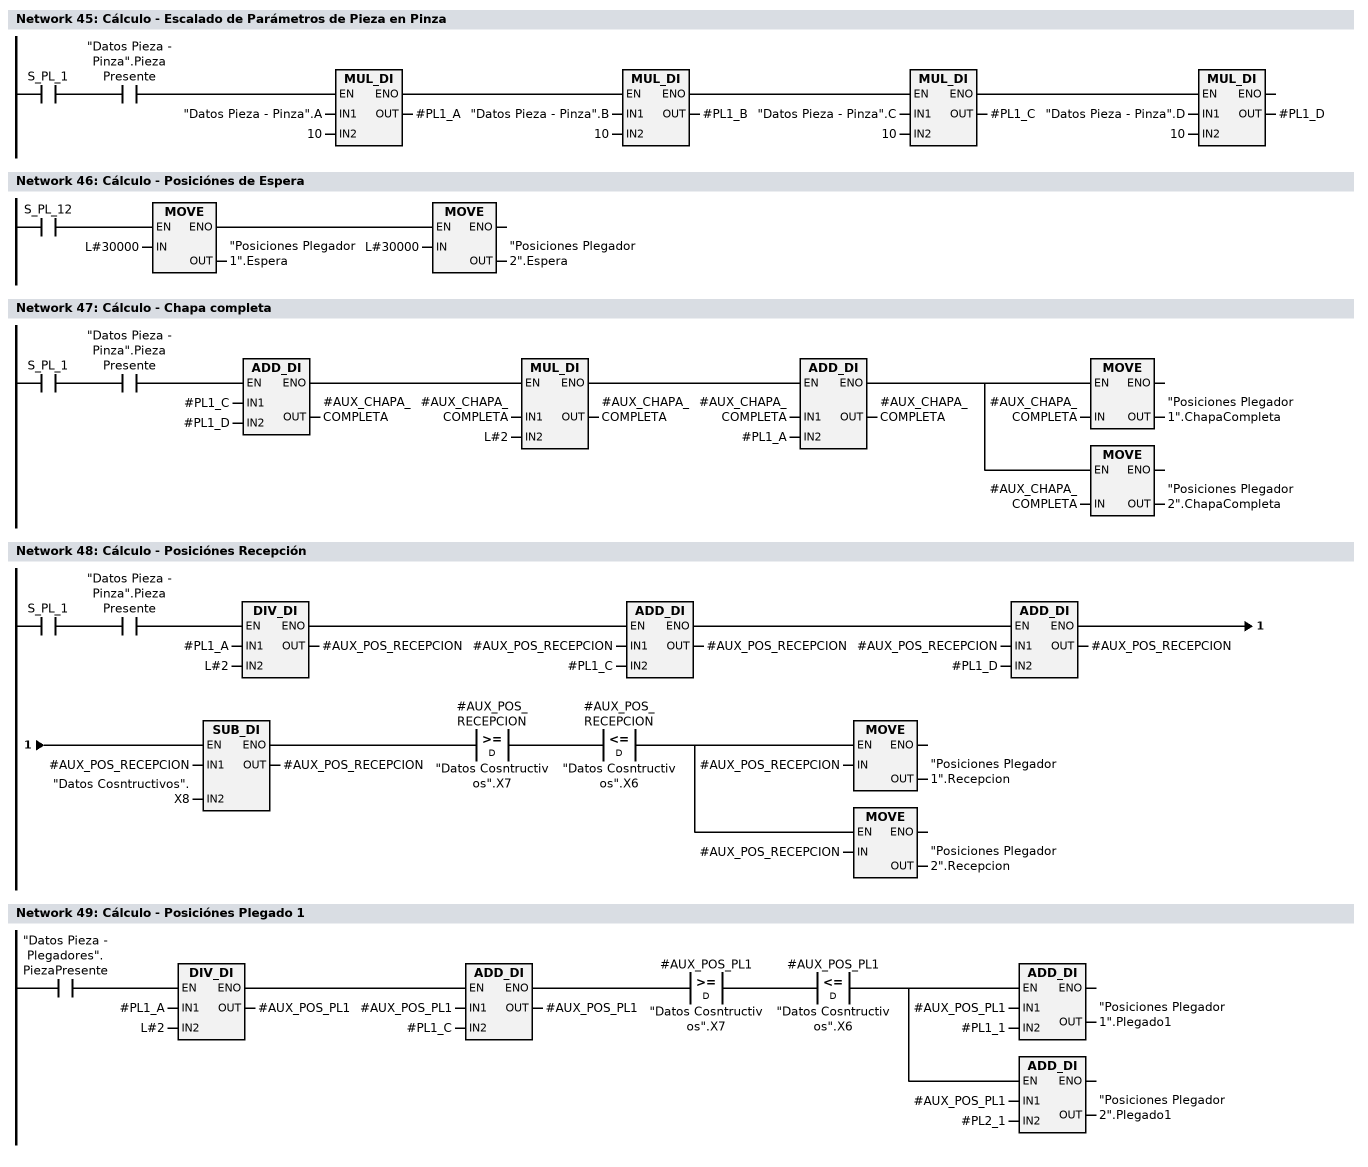
NETWORK
TITLE = Cálculo - Escalado de Parámetros de Pieza en Pinza
      A(;
      A(;
      A(;
      A     "S_PL_1";
      A     "Datos Pieza - Pinza".PiezaPresente;
      JNB   _025;
      L     "Datos Pieza - Pinza".A;
      L     10;
      *D;
      T     #PL1_A;
      AN    OV;
      SAVE;
      CLR;
_025: A     BR;
      );
      JNB   _026;
      L     "Datos Pieza - Pinza".B;
      L     10;
      *D;
      T     #PL1_B;
      AN    OV;
      SAVE;
      CLR;
_026: A     BR;
      );
      JNB   _027;
      L     "Datos Pieza - Pinza".C;
      L     10;
      *D;
      T     #PL1_C;
      AN    OV;
      SAVE;
      CLR;
_027: A     BR;
      );
      JNB   _028;
      L     "Datos Pieza - Pinza".D;
      L     10;
      *D;
      T     #PL1_D;
_028: NOP   0;
NETWORK
TITLE = Cálculo - Posiciónes de Espera
      A(;
      A     "S_PL_12";
      JNB   _029;
      L     L#30000;
      T     "Posiciones Plegador 1".Espera;
      SET;
      SAVE;
      CLR;
_029: A     BR;
      );
      JNB   _02a;
      L     L#30000;
      T     "Posiciones Plegador 2".Espera;
_02a: NOP   0;
NETWORK
TITLE = Cálculo - Chapa completa 
      A(;
      A(;
      A     "S_PL_1";
      A     "Datos Pieza - Pinza".PiezaPresente;
      JNB   _02b;
      L     #PL1_C;
      L     #PL1_D;
      +D;
      T     #AUX_CHAPA_COMPLETA;
      AN    OV;
      SAVE;
      CLR;
_02b: A     BR;
      );
      JNB   _02c;
      L     #AUX_CHAPA_COMPLETA;
      L     L#2;
      *D;
      T     #AUX_CHAPA_COMPLETA;
      AN    OV;
      SAVE;
      CLR;
_02c: A     BR;
      );
      JNB   _02d;
      L     #AUX_CHAPA_COMPLETA;
      L     #PL1_A;
      +D;
      T     #AUX_CHAPA_COMPLETA;
      AN    OV;
      SAVE;
      CLR;
_02d: A     BR;
      =     L 98.0;
      A     L 98.0;
      JNB   _02e;
      L     #AUX_CHAPA_COMPLETA;
      T     "Posiciones Plegador 1".ChapaCompleta;
_02e: NOP   0;
      A     L 98.0;
      JNB   _02f;
      L     #AUX_CHAPA_COMPLETA;
      T     "Posiciones Plegador 2".ChapaCompleta;
_02f: NOP   0;
NETWORK
TITLE = Cálculo - Posiciónes Recepción 
      A(;
      A(;
      A(;
      A(;
      A     "S_PL_1";
      A     "Datos Pieza - Pinza".PiezaPresente;
      JNB   _030;
      L     #PL1_A;
      L     L#2;
      /D;
      T     #AUX_POS_RECEPCION;
      AN    OV;
      SAVE;
      CLR;
_030: A     BR;
      );
      JNB   _031;
      L     #AUX_POS_RECEPCION;
      L     #PL1_C;
      +D;
      T     #AUX_POS_RECEPCION;
      AN    OV;
      SAVE;
      CLR;
_031: A     BR;
      );
      JNB   _032;
      L     #AUX_POS_RECEPCION;
      L     #PL1_D;
      +D;
      T     #AUX_POS_RECEPCION;
      AN    OV;
      SAVE;
      CLR;
_032: A     BR;
      );
      JNB   _033;
      L     #AUX_POS_RECEPCION;
      L     "Datos Cosntructivos".X8;
      -D;
      T     #AUX_POS_RECEPCION;
      AN    OV;
      SAVE;
      CLR;
_033: A     BR;
      );
      A(;
      L     #AUX_POS_RECEPCION;
      L     "Datos Cosntructivos".X7;
      >=D;
      );
      A(;
      L     #AUX_POS_RECEPCION;
      L     "Datos Cosntructivos".X6;
      <=D;
      );
      =     L 98.0;
      A     L 98.0;
      JNB   _034;
      L     #AUX_POS_RECEPCION;
      T     "Posiciones Plegador 1".Recepcion;
_034: NOP   0;
      A     L 98.0;
      JNB   _035;
      L     #AUX_POS_RECEPCION;
      T     "Posiciones Plegador 2".Recepcion;
_035: NOP   0;
NETWORK
TITLE = Cálculo - Posiciónes Plegado 1 
      A(;
      A(;
      A     "Datos Pieza - Plegadores".PiezaPresente;
      JNB   _036;
      L     #PL1_A;
      L     L#2;
      /D;
      T     #AUX_POS_PL1;
      AN    OV;
      SAVE;
      CLR;
_036: A     BR;
      );
      JNB   _037;
      L     #AUX_POS_PL1;
      L     #PL1_C;
      +D;
      T     #AUX_POS_PL1;
      AN    OV;
      SAVE;
      CLR;
_037: A     BR;
      );
      A(;
      L     #AUX_POS_PL1;
      L     "Datos Cosntructivos".X7;
      >=D;
      );
      A(;
      L     #AUX_POS_PL1;
      L     "Datos Cosntructivos".X6;
      <=D;
      );
      =     L 98.0;
      A     L 98.0;
      JNB   _038;
      L     #AUX_POS_PL1;
      L     #PL1_1;
      +D;
      T     "Posiciones Plegador 1".Plegado1;
_038: NOP   0;
      A     L 98.0;
      JNB   _039;
      L     #AUX_POS_PL1;
      L     #PL2_1;
      +D;
      T     "Posiciones Plegador 2".Plegado1;
_039: NOP   0;
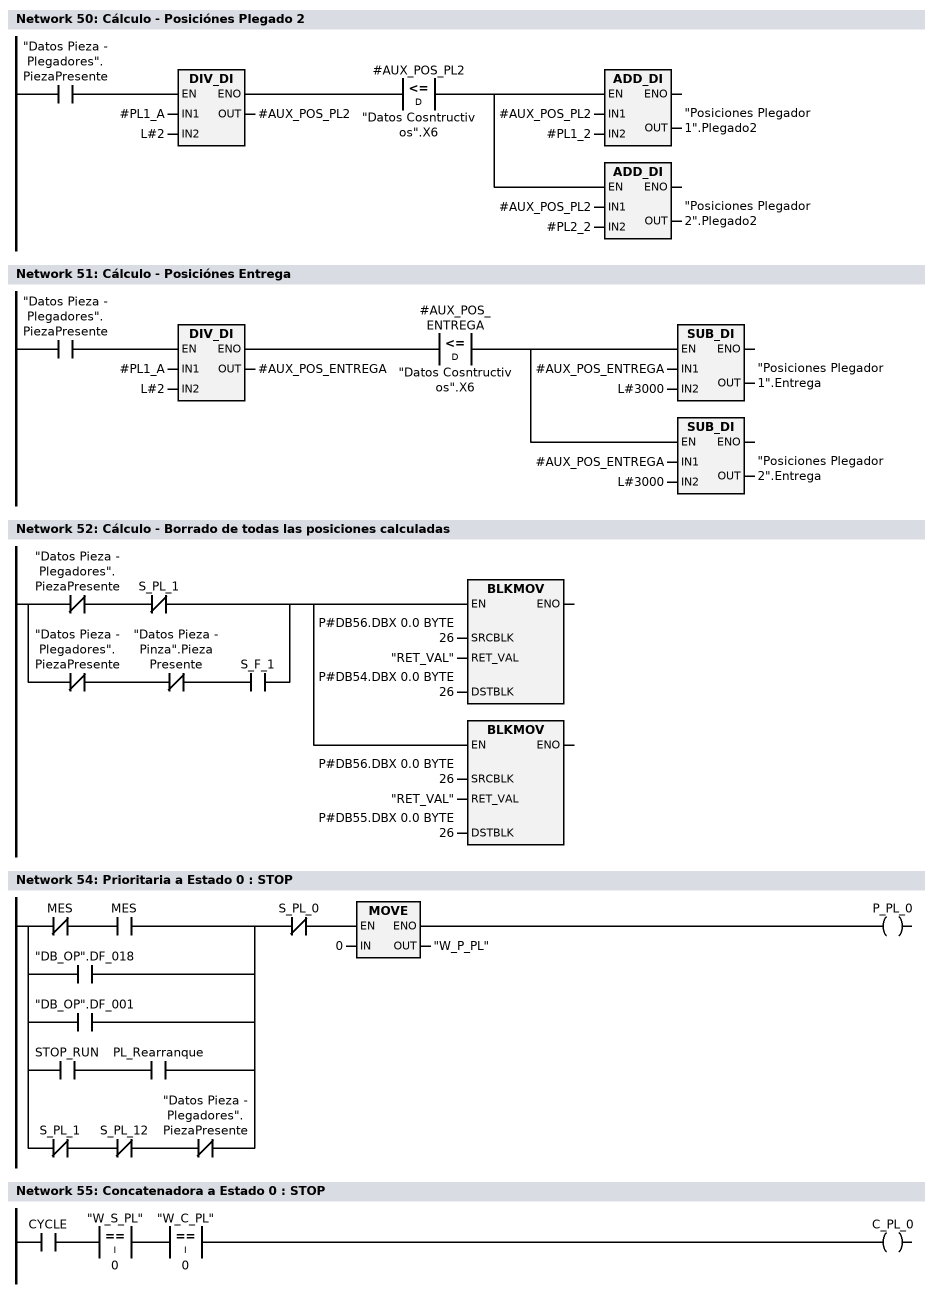
NETWORK
TITLE = Cálculo - Posiciónes Plegado 2
      A(;
      A     "Datos Pieza - Plegadores".PiezaPresente;
      JNB   _03a;
      L     #PL1_A;
      L     L#2;
      /D;
      T     #AUX_POS_PL2;
      AN    OV;
      SAVE;
      CLR;
_03a: A     BR;
      );
      A(;
      L     #AUX_POS_PL2;
      L     "Datos Cosntructivos".X6;
      <=D;
      );
      =     L 98.0;
      A     L 98.0;
      JNB   _03b;
      L     #AUX_POS_PL2;
      L     #PL1_2;
      +D;
      T     "Posiciones Plegador 1".Plegado2;
_03b: NOP   0;
      A     L 98.0;
      JNB   _03c;
      L     #AUX_POS_PL2;
      L     #PL2_2;
      +D;
      T     "Posiciones Plegador 2".Plegado2;
_03c: NOP   0;
NETWORK
TITLE = Cálculo - Posiciónes Entrega
      A(;
      A     "Datos Pieza - Plegadores".PiezaPresente;
      JNB   _03d;
      L     #PL1_A;
      L     L#2;
      /D;
      T     #AUX_POS_ENTREGA;
      AN    OV;
      SAVE;
      CLR;
_03d: A     BR;
      );
      A(;
      L     #AUX_POS_ENTREGA;
      L     "Datos Cosntructivos".X6;
      <=D;
      );
      =     L 98.0;
      A     L 98.0;
      JNB   _03e;
      L     #AUX_POS_ENTREGA;
      L     L#3000;
      -D;
      T     "Posiciones Plegador 1".Entrega;
_03e: NOP   0;
      A     L 98.0;
      JNB   _03f;
      L     #AUX_POS_ENTREGA;
      L     L#3000;
      -D;
      T     "Posiciones Plegador 2".Entrega;
_03f: NOP   0;
NETWORK
TITLE = Cálculo - Borrado de todas las posiciones calculadas 
      AN    "Datos Pieza - Plegadores".PiezaPresente;
      AN    "S_PL_1";
      O;
      AN    "Datos Pieza - Plegadores".PiezaPresente;
      AN    "Datos Pieza - Pinza".PiezaPresente;
      A     "S_F_1";
      =     L 98.0;
      A     L 98.0;
      JNB   _040;
      CALL  "BLKMOV" (
           SRCBLK                   := P#DB56.DBX 0.0 BYTE 26,
           RET_VAL                  := "RET_VAL",
           DSTBLK                   := P#DB54.DBX 0.0 BYTE 26);
_040: NOP   0;
      A     L 98.0;
      JNB   _041;
      CALL  "BLKMOV" (
           SRCBLK                   := P#DB56.DBX 0.0 BYTE 26,
           RET_VAL                  := "RET_VAL",
           DSTBLK                   := P#DB55.DBX 0.0 BYTE 26);
_041: NOP   0;
NETWORK
TITLE = ---------- CÁLCULO DE TRANSICIONES ------------
NETWORK
TITLE = Prioritaria a Estado 0 : STOP
      A(;
      AN    "MES";
      A     "MES";
      O     "DB_OP".DF_018;
      O     "DB_OP".DF_001;
      O;
      A     "STOP_RUN";
      A     "PL_Rearranque";
      O;
      AN    "S_PL_1";
      AN    "S_PL_12";
      AN    "Datos Pieza - Plegadores".PiezaPresente;
      );
      AN    "S_PL_0";
      JNB   _042;
      L     0;
      T     "W_P_PL";
      SET;
      SAVE;
      CLR;
_042: A     BR;
      =     "P_PL_0";
NETWORK
TITLE = Concatenadora a Estado 0 : STOP
      A     "CYCLE";
      A(;
      L     "W_S_PL";
      L     0;
      ==I;
      );
      A(;
      L     "W_C_PL";
      L     0;
      ==I;
      );
      =     "C_PL_0";
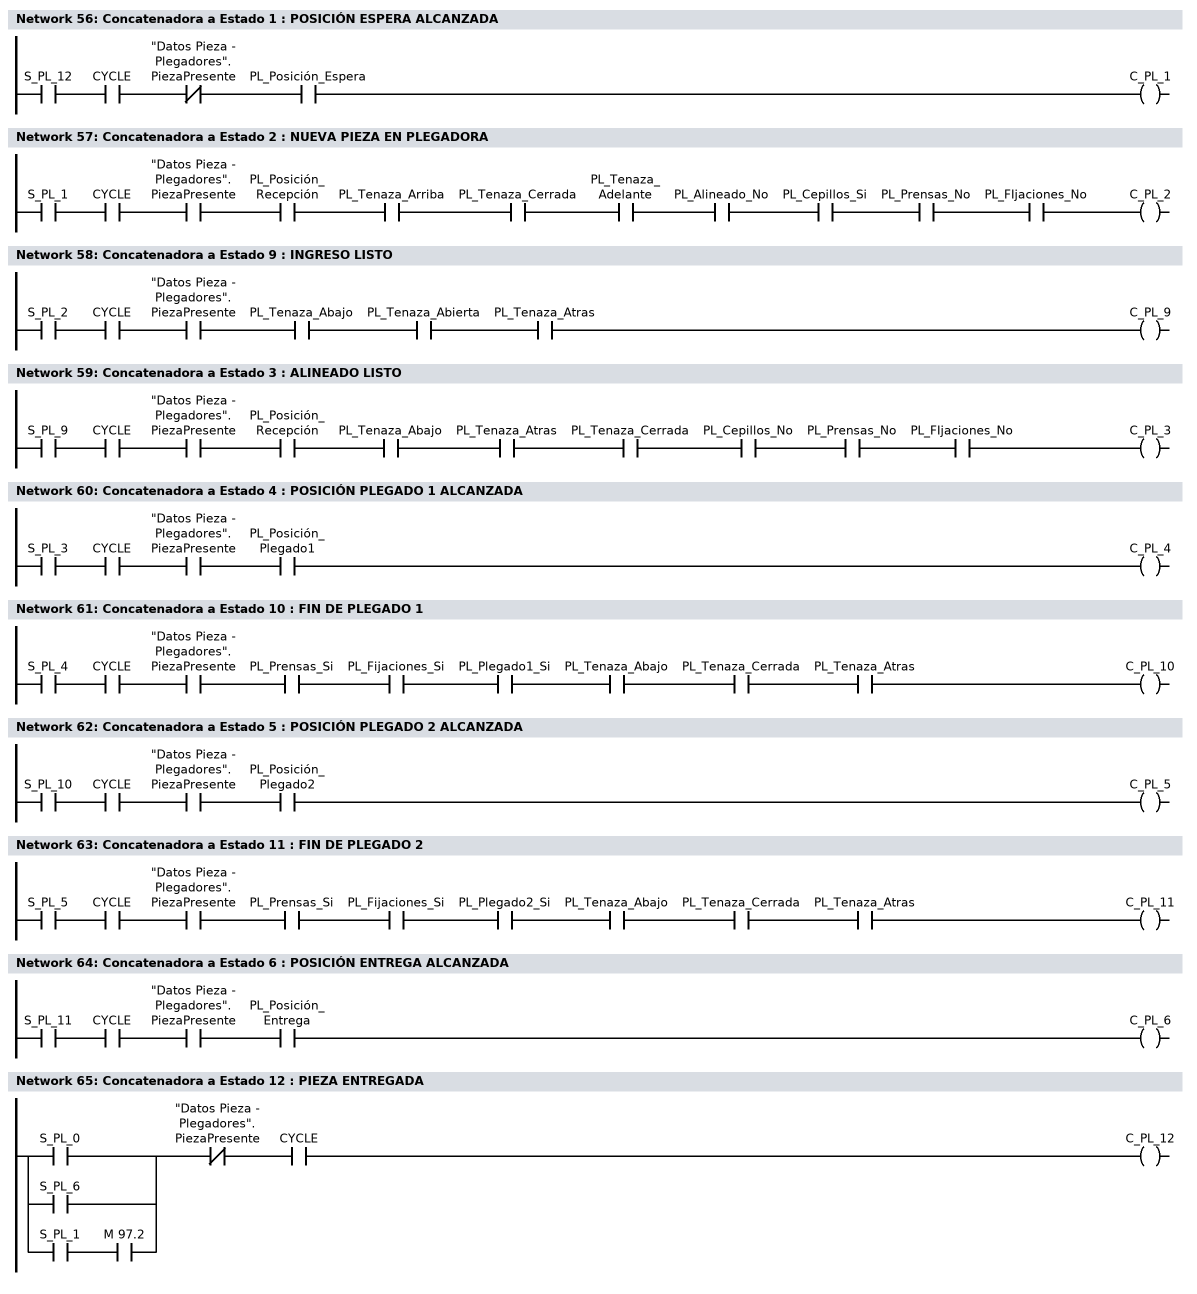
NETWORK
TITLE = Concatenadora a Estado 1 : POSICIÓN ESPERA ALCANZADA
      A     "S_PL_12";
      A     "CYCLE";
      AN    "Datos Pieza - Plegadores".PiezaPresente;
      A     "PL_Posición_Espera";
      =     "C_PL_1";
NETWORK
TITLE = Concatenadora a Estado 2 : NUEVA PIEZA EN PLEGADORA
      A     "S_PL_1";
      A     "CYCLE";
      A     "Datos Pieza - Plegadores".PiezaPresente;
      A     "PL_Posición_Recepción";
      A     "PL_Tenaza_Arriba";
      A     "PL_Tenaza_Cerrada";
      A     "PL_Tenaza_Adelante";
      A     "PL_Alineado_No";
      A     "PL_Cepillos_Si";
      A     "PL_Prensas_No";
      A     "PL_FIjaciones_No";
      =     "C_PL_2";
NETWORK
TITLE = Concatenadora a Estado 9 : INGRESO LISTO
      A     "S_PL_2";
      A     "CYCLE";
      A     "Datos Pieza - Plegadores".PiezaPresente;
      A     "PL_Tenaza_Abajo";
      A     "PL_Tenaza_Abierta";
      A     "PL_Tenaza_Atras";
      =     "C_PL_9";
NETWORK
TITLE = Concatenadora a Estado 3 : ALINEADO LISTO
      A     "S_PL_9";
      A     "CYCLE";
      A     "Datos Pieza - Plegadores".PiezaPresente;
      A     "PL_Posición_Recepción";
      A     "PL_Tenaza_Abajo";
      A     "PL_Tenaza_Atras";
      A     "PL_Tenaza_Cerrada";
      A     "PL_Cepillos_No";
      A     "PL_Prensas_No";
      A     "PL_FIjaciones_No";
      =     "C_PL_3";
NETWORK
TITLE = Concatenadora a Estado 4 : POSICIÓN PLEGADO 1 ALCANZADA
      A     "S_PL_3";
      A     "CYCLE";
      A     "Datos Pieza - Plegadores".PiezaPresente;
      A     "PL_Posición_Plegado1";
      =     "C_PL_4";
NETWORK
TITLE = Concatenadora a Estado 10 : FIN DE PLEGADO 1
      A     "S_PL_4";
      A     "CYCLE";
      A     "Datos Pieza - Plegadores".PiezaPresente;
      A     "PL_Prensas_Si";
      A     "PL_Fijaciones_Si";
      A     "PL_Plegado1_Si";
      A     "PL_Tenaza_Abajo";
      A     "PL_Tenaza_Cerrada";
      A     "PL_Tenaza_Atras";
      =     "C_PL_10";
NETWORK
TITLE = Concatenadora a Estado 5 : POSICIÓN PLEGADO 2 ALCANZADA
      A     "S_PL_10";
      A     "CYCLE";
      A     "Datos Pieza - Plegadores".PiezaPresente;
      A     "PL_Posición_Plegado2";
      =     "C_PL_5";
NETWORK
TITLE = Concatenadora a Estado 11 : FIN DE PLEGADO 2
      A     "S_PL_5";
      A     "CYCLE";
      A     "Datos Pieza - Plegadores".PiezaPresente;
      A     "PL_Prensas_Si";
      A     "PL_Fijaciones_Si";
      A     "PL_Plegado2_Si";
      A     "PL_Tenaza_Abajo";
      A     "PL_Tenaza_Cerrada";
      A     "PL_Tenaza_Atras";
      =     "C_PL_11";
NETWORK
TITLE = Concatenadora a Estado 6 : POSICIÓN ENTREGA ALCANZADA
      A     "S_PL_11";
      A     "CYCLE";
      A     "Datos Pieza - Plegadores".PiezaPresente;
      A     "PL_Posición_Entrega";
      =     "C_PL_6";
NETWORK
TITLE = Concatenadora a Estado 12 : PIEZA ENTREGADA
      A(;
      O     "S_PL_0";
      O     "S_PL_6";
      O;
      A     "S_PL_1";
      A     M 97.2;
      );
      AN    "Datos Pieza - Plegadores".PiezaPresente;
      A     "CYCLE";
      =     "C_PL_12";
NETWORK
TITLE = ------------ REARRANQUE DE PLC ----------------
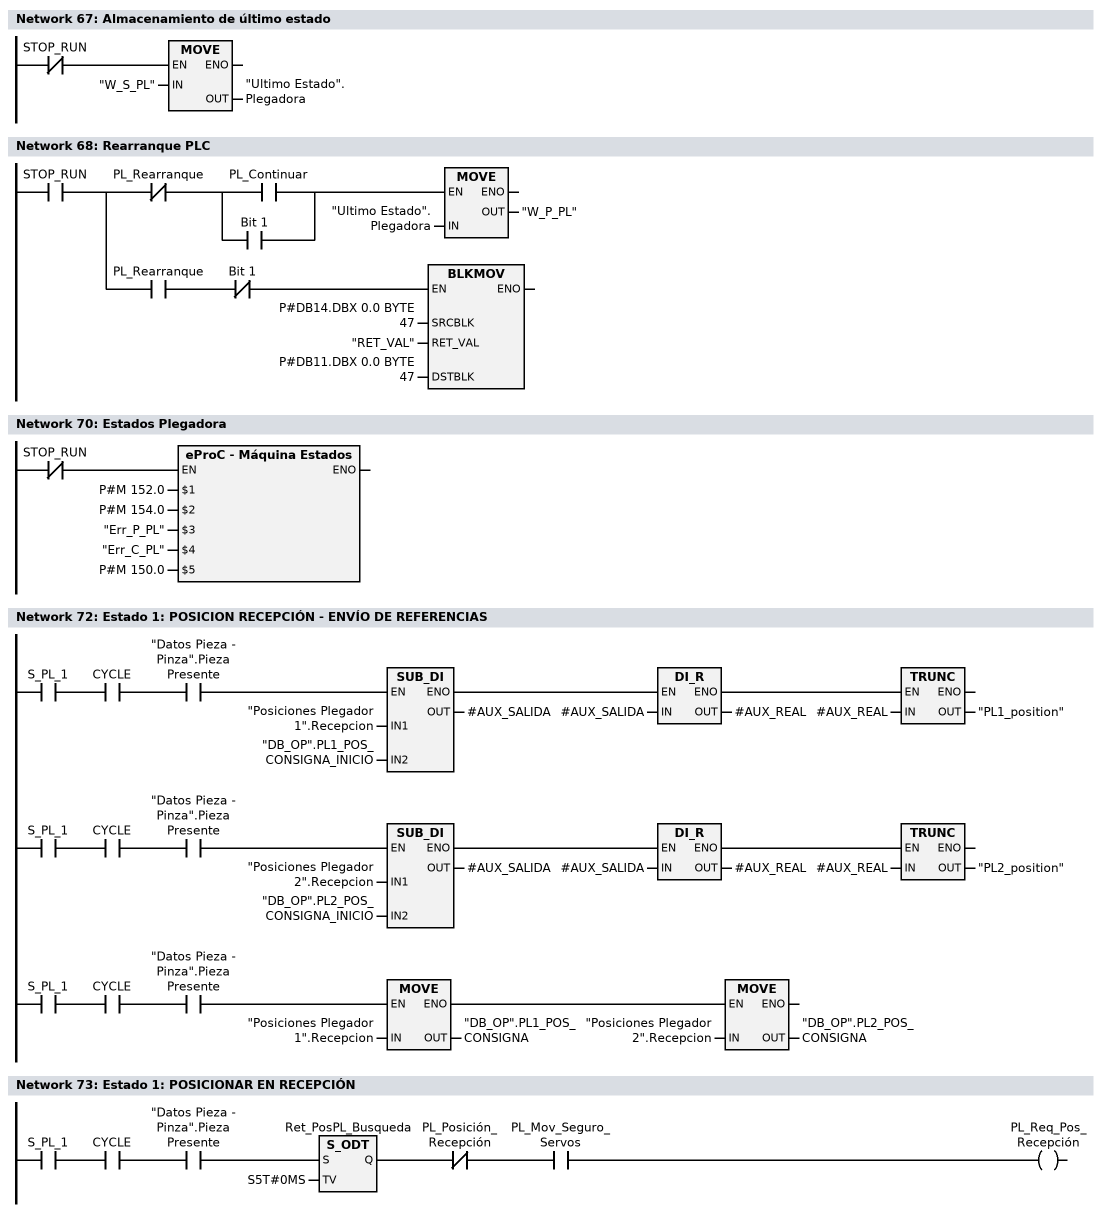
NETWORK
TITLE = Almacenamiento de último estado
      AN    "STOP_RUN";
      JNB   _043;
      L     "W_S_PL";
      T     "Ultimo Estado".Plegadora;
_043: NOP   0;
NETWORK
TITLE = Rearranque PLC
      A     "STOP_RUN";
      =     L 98.0;
      A     L 98.0;
      AN    "PL_Rearranque";
      A(;
      O     "PL_Continuar";
      O     "Bit 1";
      );
      JNB   _044;
      L     "Ultimo Estado".Plegadora;
      T     "W_P_PL";
_044: NOP   0;
      A     L 98.0;
      A     "PL_Rearranque";
      AN    "Bit 1";
      JNB   _045;
      CALL  "BLKMOV" (
           SRCBLK                   := P#DB14.DBX 0.0 BYTE 47,
           RET_VAL                  := "RET_VAL",
           DSTBLK                   := P#DB11.DBX 0.0 BYTE 47);
_045: NOP   0;
NETWORK
TITLE = ----------- MÁQUINA DE ESTADOS ----------------
NETWORK
TITLE = Estados Plegadora
      AN    "STOP_RUN";
      JNB   _046;
      CALL  "eProC - Máquina Estados" (
           $1                       := P#M 152.0,
           $2                       := P#M 154.0,
           $3                       := "Err_P_PL",
           $4                       := "Err_C_PL",
           $5                       := P#M 150.0);
_046: NOP   0;
NETWORK
TITLE = --------- GENERACIÓN DE INSTRUCCIONES ----------
NETWORK
TITLE = Estado 1: POSICION RECEPCIÓN - ENVÍO DE REFERENCIAS
      A     "S_PL_1";
      A     "CYCLE";
      A     "Datos Pieza - Pinza".PiezaPresente;
      =     L 98.0;
      A(;
      A(;
      A     L 98.0;
      JNB   _047;
      L     "Posiciones Plegador 1".Recepcion;
      L     "DB_OP".PL1_POS_CONSIGNA_INICIO;
      -D;
      T     #AUX_SALIDA;
      AN    OV;
      SAVE;
      CLR;
_047: A     BR;
      );
      JNB   _048;
      L     #AUX_SALIDA;
      DTR;
      T     #AUX_REAL;
      SET;
      SAVE;
      CLR;
_048: A     BR;
      );
      JNB   _049;
      L     #AUX_REAL;
      TRUNC;
      T     "PL1_position";
_049: NOP   0;
      A(;
      A(;
      A     L 98.0;
      JNB   _04a;
      L     "Posiciones Plegador 2".Recepcion;
      L     "DB_OP".PL2_POS_CONSIGNA_INICIO;
      -D;
      T     #AUX_SALIDA;
      AN    OV;
      SAVE;
      CLR;
_04a: A     BR;
      );
      JNB   _04b;
      L     #AUX_SALIDA;
      DTR;
      T     #AUX_REAL;
      SET;
      SAVE;
      CLR;
_04b: A     BR;
      );
      JNB   _04c;
      L     #AUX_REAL;
      TRUNC;
      T     "PL2_position";
_04c: NOP   0;
      A(;
      A     L 98.0;
      JNB   _04d;
      L     "Posiciones Plegador 1".Recepcion;
      T     "DB_OP".PL1_POS_CONSIGNA;
      SET;
      SAVE;
      CLR;
_04d: A     BR;
      );
      JNB   _04e;
      L     "Posiciones Plegador 2".Recepcion;
      T     "DB_OP".PL2_POS_CONSIGNA;
_04e: NOP   0;
NETWORK
TITLE = Estado 1: POSICIONAR EN RECEPCIÓN
      A(;
      A     "S_PL_1";
      A     "CYCLE";
      A     "Datos Pieza - Pinza".PiezaPresente;
      L     S5T#0MS;
      SD    "Ret_PosPL_Busqueda";
      NOP   0;
      NOP   0;
      NOP   0;
      A     "Ret_PosPL_Busqueda";
      );
      AN    "PL_Posición_Recepción";
      A     "PL_Mov_Seguro_Servos";
      =     "PL_Req_Pos_Recepción";
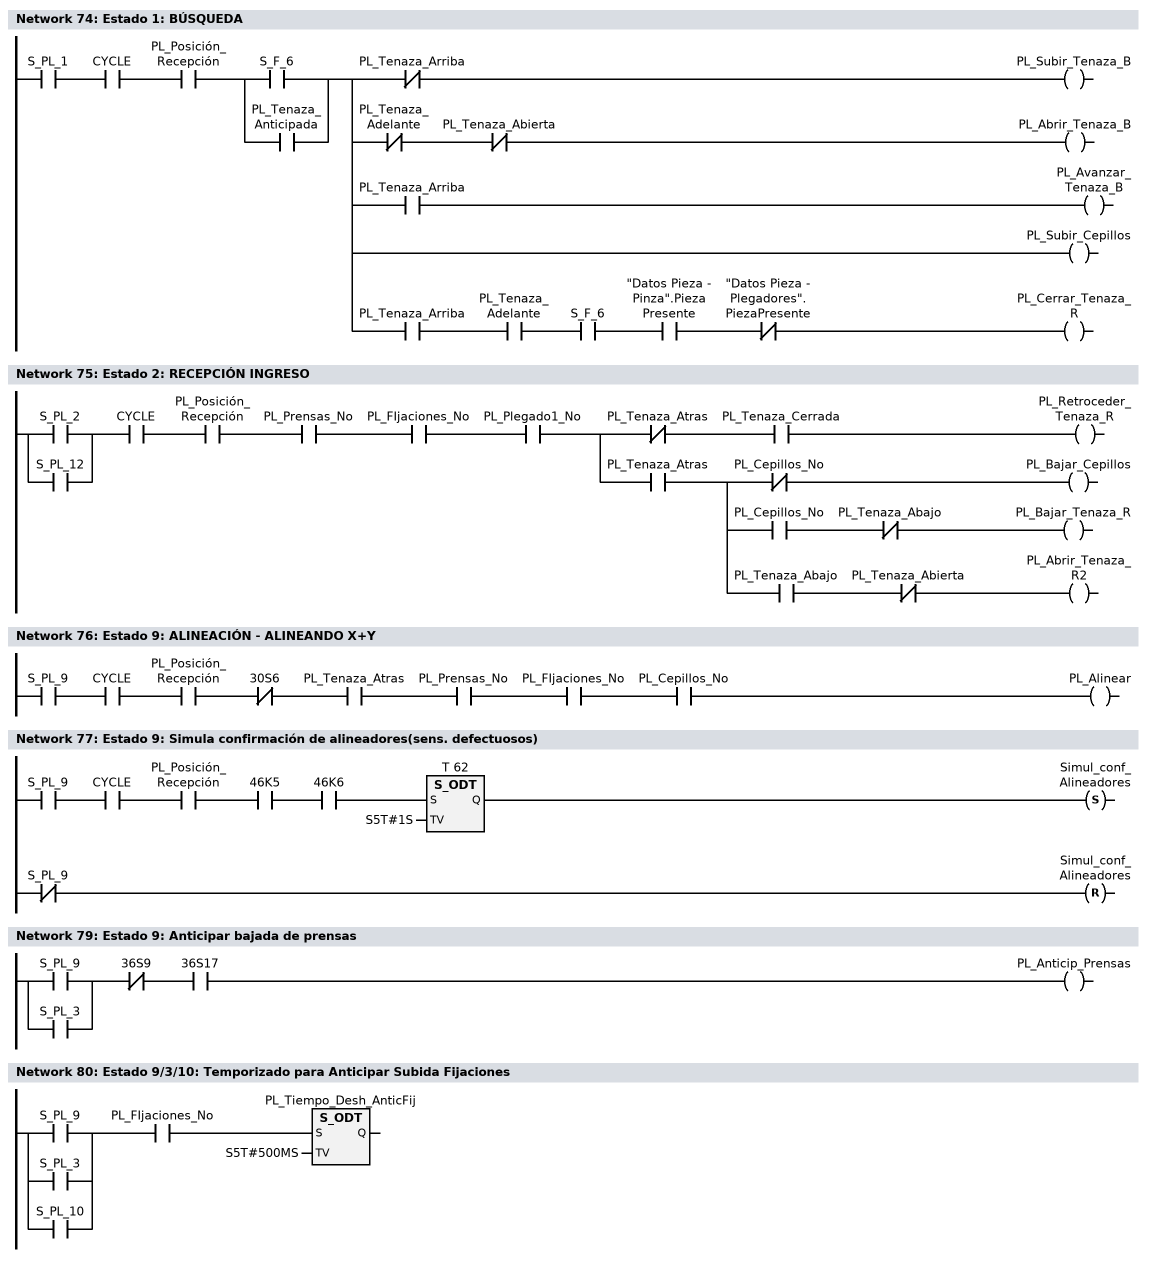
NETWORK
TITLE = Estado 1: BÚSQUEDA 
      A     "S_PL_1";
      A     "CYCLE";
      A     "PL_Posición_Recepción";
      A(;
      O     "S_F_6";
      O     "PL_Tenaza_Anticipada";
      );
      =     L 98.0;
      A     L 98.0;
      AN    "PL_Tenaza_Arriba";
      =     "PL_Subir_Tenaza_B";
      A     L 98.0;
      AN    "PL_Tenaza_Adelante";
      AN    "PL_Tenaza_Abierta";
      =     "PL_Abrir_Tenaza_B";
      A     L 98.0;
      A     "PL_Tenaza_Arriba";
      =     "PL_Avanzar_Tenaza_B";
      A     L 98.0;
      BLD   102;
      =     "PL_Subir_Cepillos";
      A     L 98.0;
      A     "PL_Tenaza_Arriba";
      A     "PL_Tenaza_Adelante";
      A     "S_F_6";
      A     "Datos Pieza - Pinza".PiezaPresente;
      AN    "Datos Pieza - Plegadores".PiezaPresente;
      =     "PL_Cerrar_Tenaza_R";
NETWORK
TITLE = Estado 2: RECEPCIÓN INGRESO
      A(;
      O     "S_PL_2";
      O     "S_PL_12";
      );
      A     "CYCLE";
      A     "PL_Posición_Recepción";
      A     "PL_Prensas_No";
      A     "PL_FIjaciones_No";
      A     "PL_Plegado1_No";
      =     L 98.0;
      A     L 98.0;
      AN    "PL_Tenaza_Atras";
      A     "PL_Tenaza_Cerrada";
      =     "PL_Retroceder_Tenaza_R";
      A     L 98.0;
      A     "PL_Tenaza_Atras";
      =     L 98.1;
      A     L 98.1;
      AN    "PL_Cepillos_No";
      =     "PL_Bajar_Cepillos";
      A     L 98.1;
      A     "PL_Cepillos_No";
      AN    "PL_Tenaza_Abajo";
      =     "PL_Bajar_Tenaza_R";
      A     L 98.1;
      A     "PL_Tenaza_Abajo";
      AN    "PL_Tenaza_Abierta";
      =     "PL_Abrir_Tenaza_R2";
NETWORK
TITLE = Estado 9: ALINEACIÓN - ALINEANDO X+Y
      A     "S_PL_9";
      A     "CYCLE";
      A     "PL_Posición_Recepción";
      AN    "30S6";
      A     "PL_Tenaza_Atras";
      A     "PL_Prensas_No";
      A     "PL_FIjaciones_No";
      A     "PL_Cepillos_No";
      =     "PL_Alinear";
NETWORK
TITLE = Estado 9: Simula confirmación de alineadores(sens. defectuosos)
      A(;
      A     "S_PL_9";
      A     "CYCLE";
      A     "PL_Posición_Recepción";
      A     "46K5";
      A     "46K6";
      L     S5T#1S;
      SD    T 62;
      NOP   0;
      NOP   0;
      NOP   0;
      A     T 62;
      );
      S     "Simul_conf_Alineadores";
      AN    "S_PL_9";
      R     "Simul_conf_Alineadores";
      NOP   0;
NETWORK
TITLE = Estado 9: ALINEACIÓN - Cerrar Tenaza
      A(;
      O     "S_PL_3";
      O(;
      A     "S_PL_9";
      A     "PL_Alineado_Si";
      S     "Aux_CerrarTenaza";
      A     "S_PL_3";
      R     "Aux_CerrarTenaza";
      A     "Aux_CerrarTenaza";
      );
      );
      A     "CYCLE";
      AN    "PL_Tenaza_Cerrada";
      =     "PL_Cerrar_Tenaza2";
NETWORK
TITLE = Estado 9: Anticipar bajada de prensas
      A(;
      O     "S_PL_9";
      O     "S_PL_3";
      );
      AN    "36S9";
      A     "36S17";
      =     "PL_Anticip_Prensas";
NETWORK
TITLE = Estado 9/3/10: Temporizado para Anticipar Subida Fijaciones
      A(;
      O     "S_PL_9";
      O     "S_PL_3";
      O     "S_PL_10";
      );
      A     "PL_FIjaciones_No";
      L     S5T#500MS;
      SD    "PL_Tiempo_Desh_AnticFij";
      NOP   0;
      NOP   0;
      NOP   0;
      NOP   0;
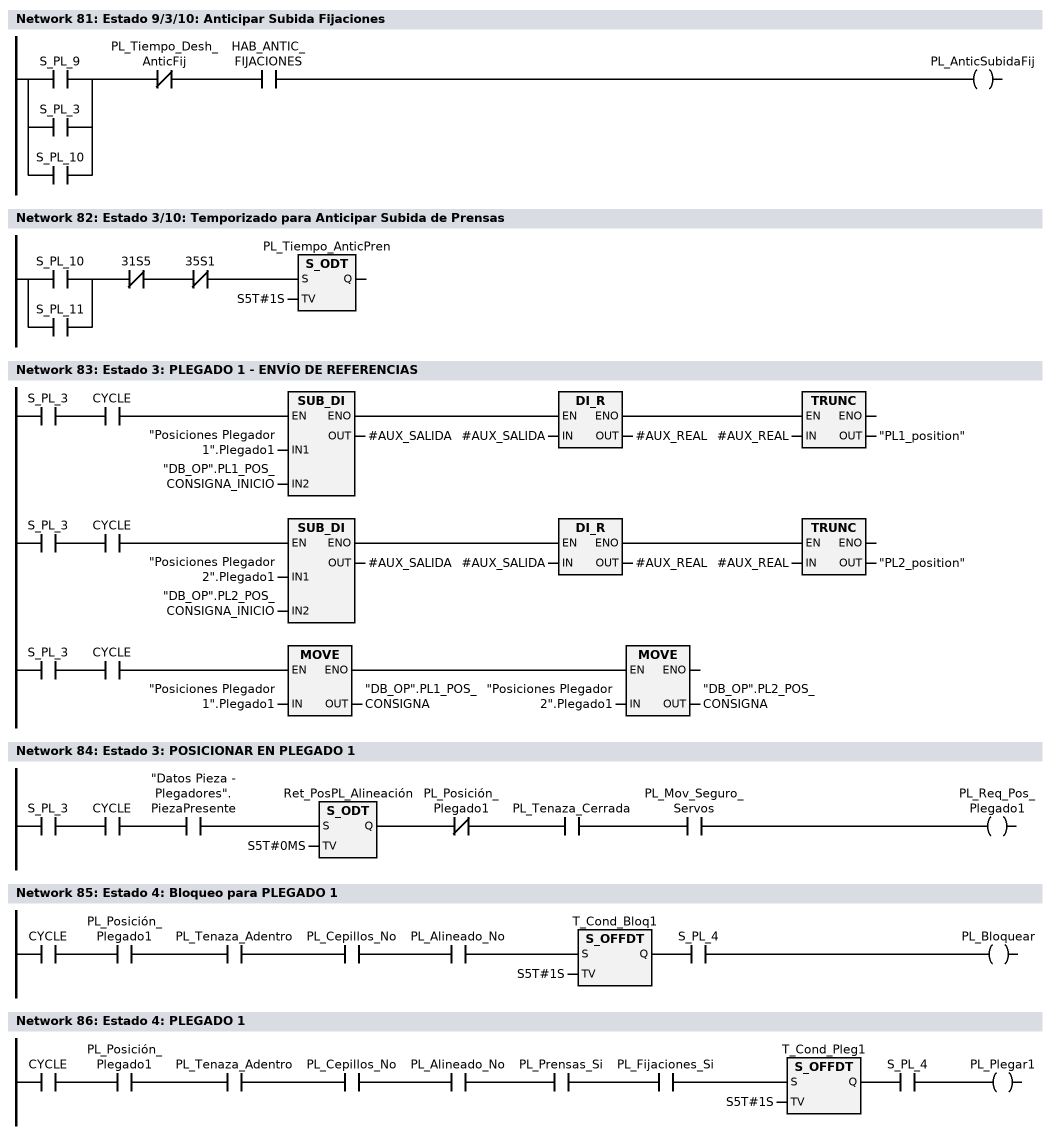
NETWORK
TITLE = Estado 9/3/10: Anticipar Subida Fijaciones
      A(;
      O     "S_PL_9";
      O     "S_PL_3";
      O     "S_PL_10";
      );
      AN    "PL_Tiempo_Desh_AnticFij";
      A     "HAB_ANTIC_FIJACIONES";
      =     "PL_AnticSubidaFij";
NETWORK
TITLE = Estado 3/10: Temporizado para Anticipar Subida de Prensas
      A(;
      O     "S_PL_10";
      O     "S_PL_11";
      );
      AN    "31S5";
      AN    "35S1";
      L     S5T#1S;
      SD    "PL_Tiempo_AnticPren";
      NOP   0;
      NOP   0;
      NOP   0;
      NOP   0;
NETWORK
TITLE = Estado 3: PLEGADO 1 - ENVÍO DE REFERENCIAS
      A     "S_PL_3";
      A     "CYCLE";
      =     L 98.0;
      A(;
      A(;
      A     L 98.0;
      JNB   _04f;
      L     "Posiciones Plegador 1".Plegado1;
      L     "DB_OP".PL1_POS_CONSIGNA_INICIO;
      -D;
      T     #AUX_SALIDA;
      AN    OV;
      SAVE;
      CLR;
_04f: A     BR;
      );
      JNB   _050;
      L     #AUX_SALIDA;
      DTR;
      T     #AUX_REAL;
      SET;
      SAVE;
      CLR;
_050: A     BR;
      );
      JNB   _051;
      L     #AUX_REAL;
      TRUNC;
      T     "PL1_position";
_051: NOP   0;
      A(;
      A(;
      A     L 98.0;
      JNB   _052;
      L     "Posiciones Plegador 2".Plegado1;
      L     "DB_OP".PL2_POS_CONSIGNA_INICIO;
      -D;
      T     #AUX_SALIDA;
      AN    OV;
      SAVE;
      CLR;
_052: A     BR;
      );
      JNB   _053;
      L     #AUX_SALIDA;
      DTR;
      T     #AUX_REAL;
      SET;
      SAVE;
      CLR;
_053: A     BR;
      );
      JNB   _054;
      L     #AUX_REAL;
      TRUNC;
      T     "PL2_position";
_054: NOP   0;
      A(;
      A     L 98.0;
      JNB   _055;
      L     "Posiciones Plegador 1".Plegado1;
      T     "DB_OP".PL1_POS_CONSIGNA;
      SET;
      SAVE;
      CLR;
_055: A     BR;
      );
      JNB   _056;
      L     "Posiciones Plegador 2".Plegado1;
      T     "DB_OP".PL2_POS_CONSIGNA;
_056: NOP   0;
NETWORK
TITLE = Estado 3: POSICIONAR EN PLEGADO 1
      A(;
      A     "S_PL_3";
      A     "CYCLE";
      A     "Datos Pieza - Plegadores".PiezaPresente;
      L     S5T#0MS;
      SD    "Ret_PosPL_Alineación";
      NOP   0;
      NOP   0;
      NOP   0;
      A     "Ret_PosPL_Alineación";
      );
      AN    "PL_Posición_Plegado1";
      A     "PL_Tenaza_Cerrada";
      A     "PL_Mov_Seguro_Servos";
      =     "PL_Req_Pos_Plegado1";
NETWORK
TITLE = Estado 4: Bloqueo para PLEGADO 1 
      A(;
      A     "CYCLE";
      A     "PL_Posición_Plegado1";
      A     "PL_Tenaza_Adentro";
      A     "PL_Cepillos_No";
      A     "PL_Alineado_No";
      L     S5T#1S;
      SF    "T_Cond_Bloq1";
      NOP   0;
      NOP   0;
      NOP   0;
      A     "T_Cond_Bloq1";
      );
      A     "S_PL_4";
      =     "PL_Bloquear";
NETWORK
TITLE = Estado 4: PLEGADO 1 
      A(;
      A     "CYCLE";
      A     "PL_Posición_Plegado1";
      A     "PL_Tenaza_Adentro";
      A     "PL_Cepillos_No";
      A     "PL_Alineado_No";
      A     "PL_Prensas_Si";
      A     "PL_Fijaciones_Si";
      L     S5T#1S;
      SF    "T_Cond_Pleg1";
      NOP   0;
      NOP   0;
      NOP   0;
      A     "T_Cond_Pleg1";
      );
      A     "S_PL_4";
      =     "PL_Plegar1";
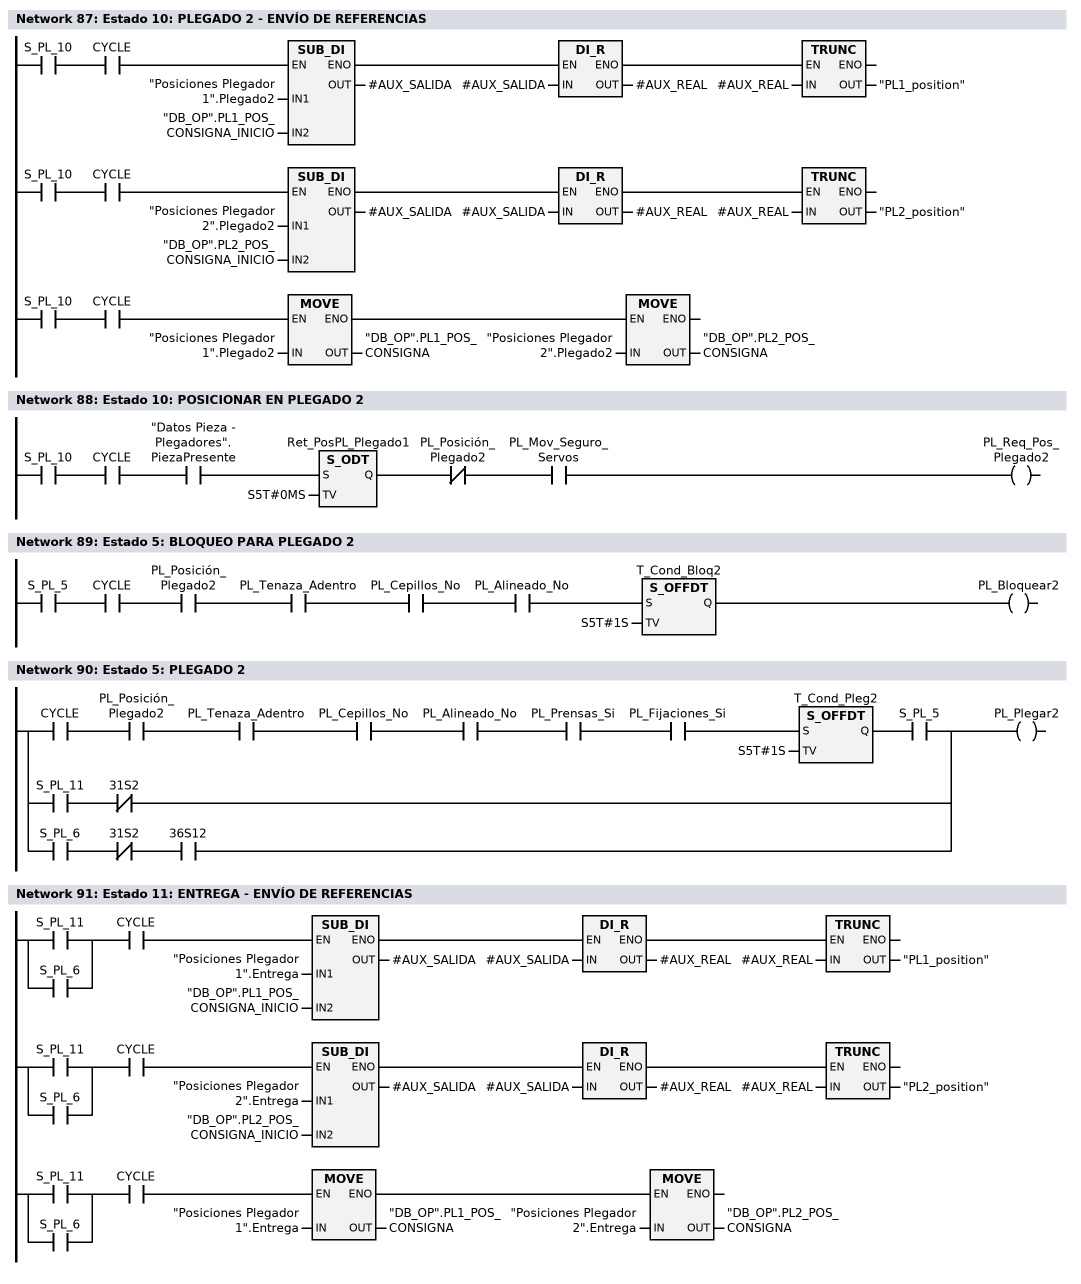
NETWORK
TITLE = Estado 10: PLEGADO 2 - ENVÍO DE REFERENCIAS
      A     "S_PL_10";
      A     "CYCLE";
      =     L 98.0;
      A(;
      A(;
      A     L 98.0;
      JNB   _057;
      L     "Posiciones Plegador 1".Plegado2;
      L     "DB_OP".PL1_POS_CONSIGNA_INICIO;
      -D;
      T     #AUX_SALIDA;
      AN    OV;
      SAVE;
      CLR;
_057: A     BR;
      );
      JNB   _058;
      L     #AUX_SALIDA;
      DTR;
      T     #AUX_REAL;
      SET;
      SAVE;
      CLR;
_058: A     BR;
      );
      JNB   _059;
      L     #AUX_REAL;
      TRUNC;
      T     "PL1_position";
_059: NOP   0;
      A(;
      A(;
      A     L 98.0;
      JNB   _05a;
      L     "Posiciones Plegador 2".Plegado2;
      L     "DB_OP".PL2_POS_CONSIGNA_INICIO;
      -D;
      T     #AUX_SALIDA;
      AN    OV;
      SAVE;
      CLR;
_05a: A     BR;
      );
      JNB   _05b;
      L     #AUX_SALIDA;
      DTR;
      T     #AUX_REAL;
      SET;
      SAVE;
      CLR;
_05b: A     BR;
      );
      JNB   _05c;
      L     #AUX_REAL;
      TRUNC;
      T     "PL2_position";
_05c: NOP   0;
      A(;
      A     L 98.0;
      JNB   _05d;
      L     "Posiciones Plegador 1".Plegado2;
      T     "DB_OP".PL1_POS_CONSIGNA;
      SET;
      SAVE;
      CLR;
_05d: A     BR;
      );
      JNB   _05e;
      L     "Posiciones Plegador 2".Plegado2;
      T     "DB_OP".PL2_POS_CONSIGNA;
_05e: NOP   0;
NETWORK
TITLE = Estado 10: POSICIONAR EN PLEGADO 2
      A(;
      A     "S_PL_10";
      A     "CYCLE";
      A     "Datos Pieza - Plegadores".PiezaPresente;
      L     S5T#0MS;
      SD    "Ret_PosPL_Plegado1";
      NOP   0;
      NOP   0;
      NOP   0;
      A     "Ret_PosPL_Plegado1";
      );
      AN    "PL_Posición_Plegado2";
      A     "PL_Mov_Seguro_Servos";
      =     "PL_Req_Pos_Plegado2";
NETWORK
TITLE = Estado 5: BLOQUEO PARA PLEGADO 2
      A     "S_PL_5";
      A     "CYCLE";
      A     "PL_Posición_Plegado2";
      A     "PL_Tenaza_Adentro";
      A     "PL_Cepillos_No";
      A     "PL_Alineado_No";
      L     S5T#1S;
      SF    "T_Cond_Bloq2";
      NOP   0;
      NOP   0;
      NOP   0;
      A     "T_Cond_Bloq2";
      =     "PL_Bloquear2";
NETWORK
TITLE = Estado 5: PLEGADO 2
      A(;
      A     "CYCLE";
      A     "PL_Posición_Plegado2";
      A     "PL_Tenaza_Adentro";
      A     "PL_Cepillos_No";
      A     "PL_Alineado_No";
      A     "PL_Prensas_Si";
      A     "PL_Fijaciones_Si";
      L     S5T#1S;
      SF    "T_Cond_Pleg2";
      NOP   0;
      NOP   0;
      NOP   0;
      A     "T_Cond_Pleg2";
      );
      A     "S_PL_5";
      O;
      A     "S_PL_11";
      AN    "31S2";
      O;
      A     "S_PL_6";
      AN    "31S2";
      A     "36S12";
      =     "PL_Plegar2";
NETWORK
TITLE = Estado 11: ENTREGA - ENVÍO DE REFERENCIAS
      A(;
      O     "S_PL_11";
      O     "S_PL_6";
      );
      A     "CYCLE";
      =     L 98.0;
      A(;
      A(;
      A     L 98.0;
      JNB   _05f;
      L     "Posiciones Plegador 1".Entrega;
      L     "DB_OP".PL1_POS_CONSIGNA_INICIO;
      -D;
      T     #AUX_SALIDA;
      AN    OV;
      SAVE;
      CLR;
_05f: A     BR;
      );
      JNB   _060;
      L     #AUX_SALIDA;
      DTR;
      T     #AUX_REAL;
      SET;
      SAVE;
      CLR;
_060: A     BR;
      );
      JNB   _061;
      L     #AUX_REAL;
      TRUNC;
      T     "PL1_position";
_061: NOP   0;
      A(;
      A(;
      A     L 98.0;
      JNB   _062;
      L     "Posiciones Plegador 2".Entrega;
      L     "DB_OP".PL2_POS_CONSIGNA_INICIO;
      -D;
      T     #AUX_SALIDA;
      AN    OV;
      SAVE;
      CLR;
_062: A     BR;
      );
      JNB   _063;
      L     #AUX_SALIDA;
      DTR;
      T     #AUX_REAL;
      SET;
      SAVE;
      CLR;
_063: A     BR;
      );
      JNB   _064;
      L     #AUX_REAL;
      TRUNC;
      T     "PL2_position";
_064: NOP   0;
      A(;
      A     L 98.0;
      JNB   _065;
      L     "Posiciones Plegador 1".Entrega;
      T     "DB_OP".PL1_POS_CONSIGNA;
      SET;
      SAVE;
      CLR;
_065: A     BR;
      );
      JNB   _066;
      L     "Posiciones Plegador 2".Entrega;
      T     "DB_OP".PL2_POS_CONSIGNA;
_066: NOP   0;
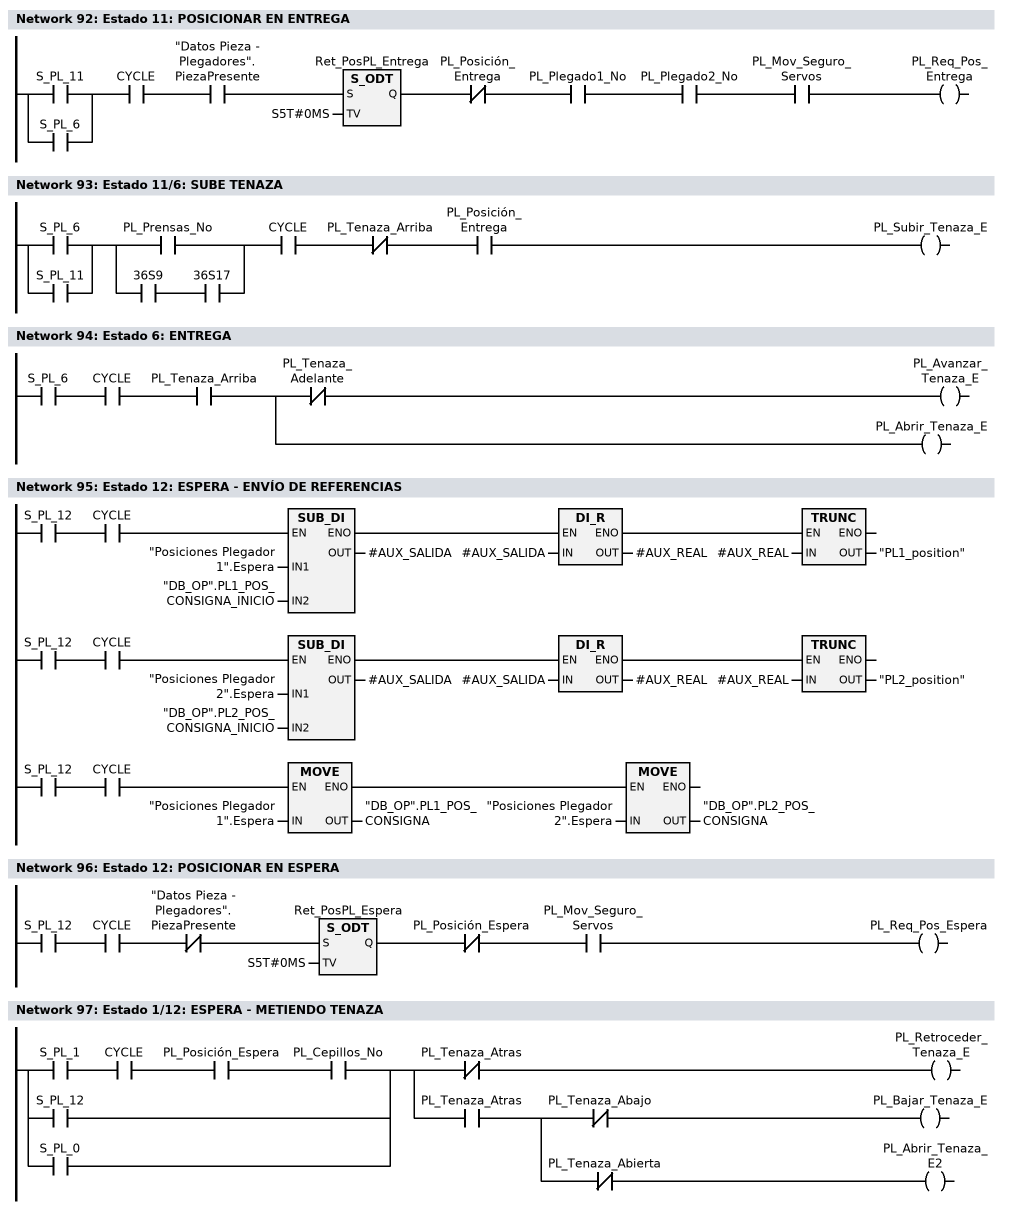
NETWORK
TITLE = Estado 11: POSICIONAR EN ENTREGA
      A(;
      A(;
      O     "S_PL_11";
      O     "S_PL_6";
      );
      A     "CYCLE";
      A     "Datos Pieza - Plegadores".PiezaPresente;
      L     S5T#0MS;
      SD    "Ret_PosPL_Entrega";
      NOP   0;
      NOP   0;
      NOP   0;
      A     "Ret_PosPL_Entrega";
      );
      AN    "PL_Posición_Entrega";
      A     "PL_Plegado1_No";
      A     "PL_Plegado2_No";
      A     "PL_Mov_Seguro_Servos";
      =     "PL_Req_Pos_Entrega";
NETWORK
TITLE = Estado 11/6: SUBE TENAZA
      A(;
      O     "S_PL_6";
      O     "S_PL_11";
      );
      A(;
      O     "PL_Prensas_No";
      O;
      A     "36S9";
      A     "36S17";
      );
      A     "CYCLE";
      AN    "PL_Tenaza_Arriba";
      A     "PL_Posición_Entrega";
      =     "PL_Subir_Tenaza_E";
NETWORK
TITLE = Estado 6: ENTREGA
      A     "S_PL_6";
      A     "CYCLE";
      A     "PL_Tenaza_Arriba";
      =     L 98.0;
      A     L 98.0;
      AN    "PL_Tenaza_Adelante";
      =     "PL_Avanzar_Tenaza_E";
      A     L 98.0;
      BLD   102;
      =     "PL_Abrir_Tenaza_E";
NETWORK
TITLE = Estado 12: ESPERA - ENVÍO DE REFERENCIAS
      A     "S_PL_12";
      A     "CYCLE";
      =     L 98.0;
      A(;
      A(;
      A     L 98.0;
      JNB   _067;
      L     "Posiciones Plegador 1".Espera;
      L     "DB_OP".PL1_POS_CONSIGNA_INICIO;
      -D;
      T     #AUX_SALIDA;
      AN    OV;
      SAVE;
      CLR;
_067: A     BR;
      );
      JNB   _068;
      L     #AUX_SALIDA;
      DTR;
      T     #AUX_REAL;
      SET;
      SAVE;
      CLR;
_068: A     BR;
      );
      JNB   _069;
      L     #AUX_REAL;
      TRUNC;
      T     "PL1_position";
_069: NOP   0;
      A(;
      A(;
      A     L 98.0;
      JNB   _06a;
      L     "Posiciones Plegador 2".Espera;
      L     "DB_OP".PL2_POS_CONSIGNA_INICIO;
      -D;
      T     #AUX_SALIDA;
      AN    OV;
      SAVE;
      CLR;
_06a: A     BR;
      );
      JNB   _06b;
      L     #AUX_SALIDA;
      DTR;
      T     #AUX_REAL;
      SET;
      SAVE;
      CLR;
_06b: A     BR;
      );
      JNB   _06c;
      L     #AUX_REAL;
      TRUNC;
      T     "PL2_position";
_06c: NOP   0;
      A(;
      A     L 98.0;
      JNB   _06d;
      L     "Posiciones Plegador 1".Espera;
      T     "DB_OP".PL1_POS_CONSIGNA;
      SET;
      SAVE;
      CLR;
_06d: A     BR;
      );
      JNB   _06e;
      L     "Posiciones Plegador 2".Espera;
      T     "DB_OP".PL2_POS_CONSIGNA;
_06e: NOP   0;
NETWORK
TITLE = Estado 12: POSICIONAR EN ESPERA
      A(;
      A     "S_PL_12";
      A     "CYCLE";
      AN    "Datos Pieza - Plegadores".PiezaPresente;
      L     S5T#0MS;
      SD    "Ret_PosPL_Espera";
      NOP   0;
      NOP   0;
      NOP   0;
      A     "Ret_PosPL_Espera";
      );
      AN    "PL_Posición_Espera";
      A     "PL_Mov_Seguro_Servos";
      =     "PL_Req_Pos_Espera";
NETWORK
TITLE = Estado 1/12: ESPERA - METIENDO TENAZA
      A     "S_PL_1";
      A     "CYCLE";
      A     "PL_Posición_Espera";
      A     "PL_Cepillos_No";
      O     "S_PL_12";
      O     "S_PL_0";
      =     L 98.0;
      A     L 98.0;
      AN    "PL_Tenaza_Atras";
      =     "PL_Retroceder_Tenaza_E";
      A     L 98.0;
      A     "PL_Tenaza_Atras";
      =     L 98.1;
      A     L 98.1;
      AN    "PL_Tenaza_Abajo";
      =     "PL_Bajar_Tenaza_E";
      A     L 98.1;
      AN    "PL_Tenaza_Abierta";
      =     "PL_Abrir_Tenaza_E2";
NETWORK
TITLE = -------------- ACTIVACIÓN DE SALIDAS ----------------
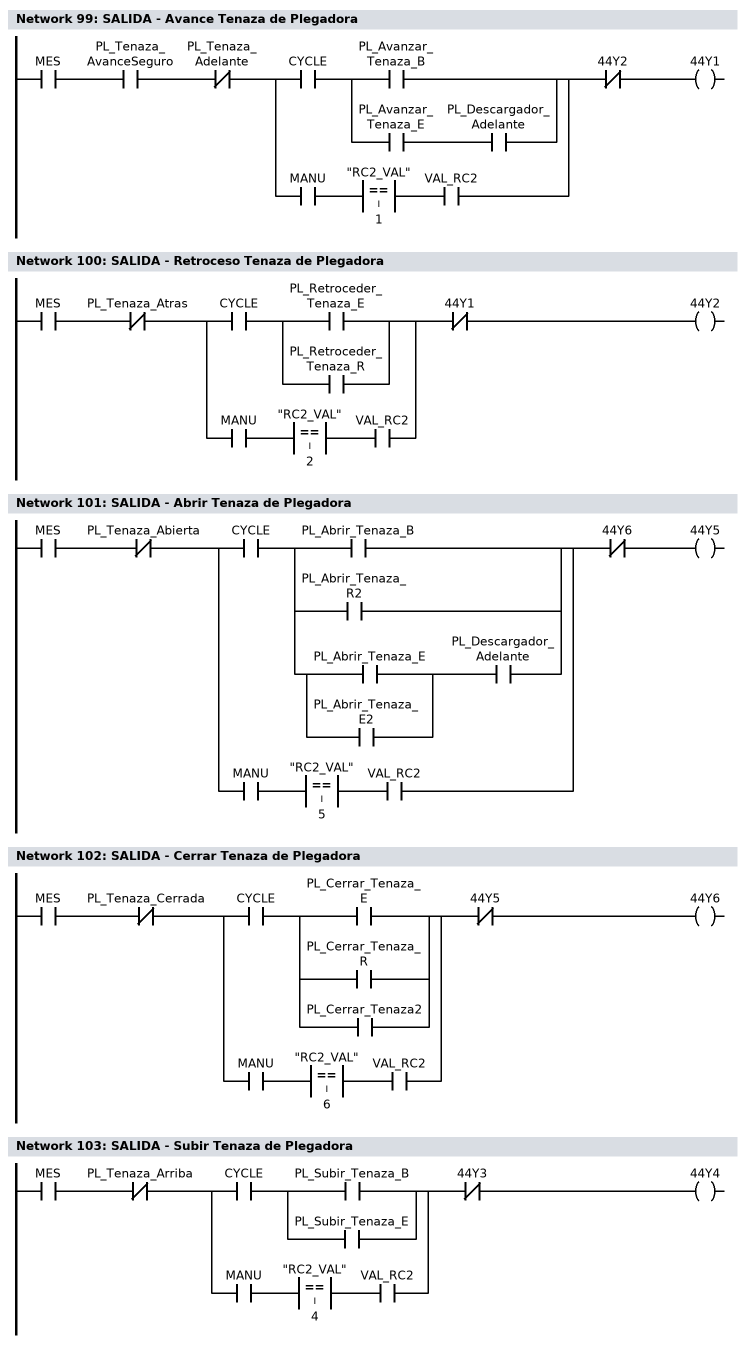
NETWORK
TITLE = SALIDA - Avance Tenaza de Plegadora
      A     "MES";
      A     "PL_Tenaza_AvanceSeguro";
      AN    "PL_Tenaza_Adelante";
      A(;
      A     "CYCLE";
      A(;
      O     "PL_Avanzar_Tenaza_B";
      O;
      A     "PL_Avanzar_Tenaza_E";
      A     "PL_Descargador_Adelante";
      );
      O;
      A     "MANU";
      A(;
      L     "RC2_VAL";
      L     1;
      ==I;
      );
      A     "VAL_RC2";
      );
      AN    "44Y2";
      =     "44Y1";
NETWORK
TITLE = SALIDA - Retroceso Tenaza de Plegadora
      A     "MES";
      AN    "PL_Tenaza_Atras";
      A(;
      A     "CYCLE";
      A(;
      O     "PL_Retroceder_Tenaza_E";
      O     "PL_Retroceder_Tenaza_R";
      );
      O;
      A     "MANU";
      A(;
      L     "RC2_VAL";
      L     2;
      ==I;
      );
      A     "VAL_RC2";
      );
      AN    "44Y1";
      =     "44Y2";
NETWORK
TITLE = SALIDA - Abrir Tenaza de Plegadora
      A     "MES";
      AN    "PL_Tenaza_Abierta";
      A(;
      A     "CYCLE";
      A(;
      O     "PL_Abrir_Tenaza_B";
      O     "PL_Abrir_Tenaza_R2";
      O;
      A(;
      O     "PL_Abrir_Tenaza_E";
      O     "PL_Abrir_Tenaza_E2";
      );
      A     "PL_Descargador_Adelante";
      );
      O;
      A     "MANU";
      A(;
      L     "RC2_VAL";
      L     5;
      ==I;
      );
      A     "VAL_RC2";
      );
      AN    "44Y6";
      =     "44Y5";
NETWORK
TITLE = SALIDA - Cerrar Tenaza de Plegadora 
      A     "MES";
      AN    "PL_Tenaza_Cerrada";
      A(;
      A     "CYCLE";
      A(;
      O     "PL_Cerrar_Tenaza_E";
      O     "PL_Cerrar_Tenaza_R";
      O     "PL_Cerrar_Tenaza2";
      );
      O;
      A     "MANU";
      A(;
      L     "RC2_VAL";
      L     6;
      ==I;
      );
      A     "VAL_RC2";
      );
      AN    "44Y5";
      =     "44Y6";
NETWORK
TITLE = SALIDA - Subir Tenaza de Plegadora
      A     "MES";
      AN    "PL_Tenaza_Arriba";
      A(;
      A     "CYCLE";
      A(;
      O     "PL_Subir_Tenaza_B";
      O     "PL_Subir_Tenaza_E";
      );
      O;
      A     "MANU";
      A(;
      L     "RC2_VAL";
      L     4;
      ==I;
      );
      A     "VAL_RC2";
      );
      AN    "44Y3";
      =     "44Y4";
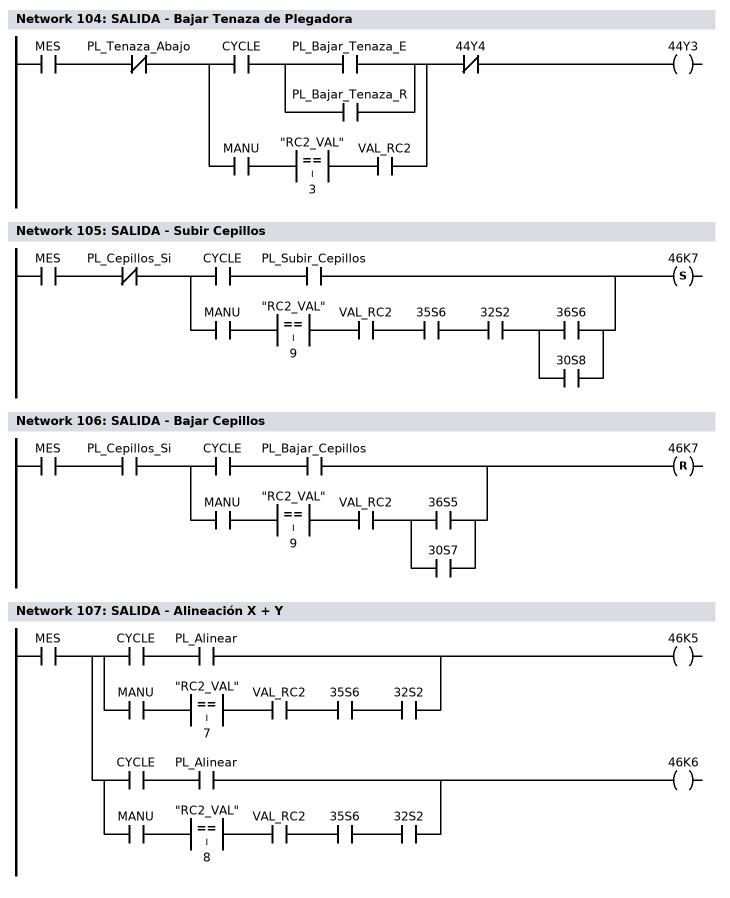
NETWORK
TITLE = SALIDA - Bajar Tenaza de Plegadora
      A     "MES";
      AN    "PL_Tenaza_Abajo";
      A(;
      A     "CYCLE";
      A(;
      O     "PL_Bajar_Tenaza_E";
      O     "PL_Bajar_Tenaza_R";
      );
      O;
      A     "MANU";
      A(;
      L     "RC2_VAL";
      L     3;
      ==I;
      );
      A     "VAL_RC2";
      );
      AN    "44Y4";
      =     "44Y3";
NETWORK
TITLE = SALIDA - Subir Cepillos
      A     "MES";
      AN    "PL_Cepillos_Si";
      A(;
      A     "CYCLE";
      A     "PL_Subir_Cepillos";
      O;
      A     "MANU";
      A(;
      L     "RC2_VAL";
      L     9;
      ==I;
      );
      A     "VAL_RC2";
      A     "35S6";
      A     "32S2";
      A(;
      O     "36S6";
      O     "30S8";
      );
      );
      S     "46K7";
NETWORK
TITLE = SALIDA - Bajar Cepillos
      A     "MES";
      A     "PL_Cepillos_Si";
      A(;
      A     "CYCLE";
      A     "PL_Bajar_Cepillos";
      O;
      A     "MANU";
      A(;
      L     "RC2_VAL";
      L     9;
      ==I;
      );
      A     "VAL_RC2";
      A(;
      O     "36S5";
      O     "30S7";
      );
      );
      R     "46K7";
NETWORK
TITLE = SALIDA - Alineación X + Y
      A     "MES";
      =     L 98.0;
      A     L 98.0;
      A(;
      A     "CYCLE";
      A     "PL_Alinear";
      O;
      A     "MANU";
      A(;
      L     "RC2_VAL";
      L     7;
      ==I;
      );
      A     "VAL_RC2";
      A     "35S6";
      A     "32S2";
      );
      =     "46K5";
      A     L 98.0;
      A(;
      A     "CYCLE";
      A     "PL_Alinear";
      O;
      A     "MANU";
      A(;
      L     "RC2_VAL";
      L     8;
      ==I;
      );
      A     "VAL_RC2";
      A     "35S6";
      A     "32S2";
      );
      =     "46K6";
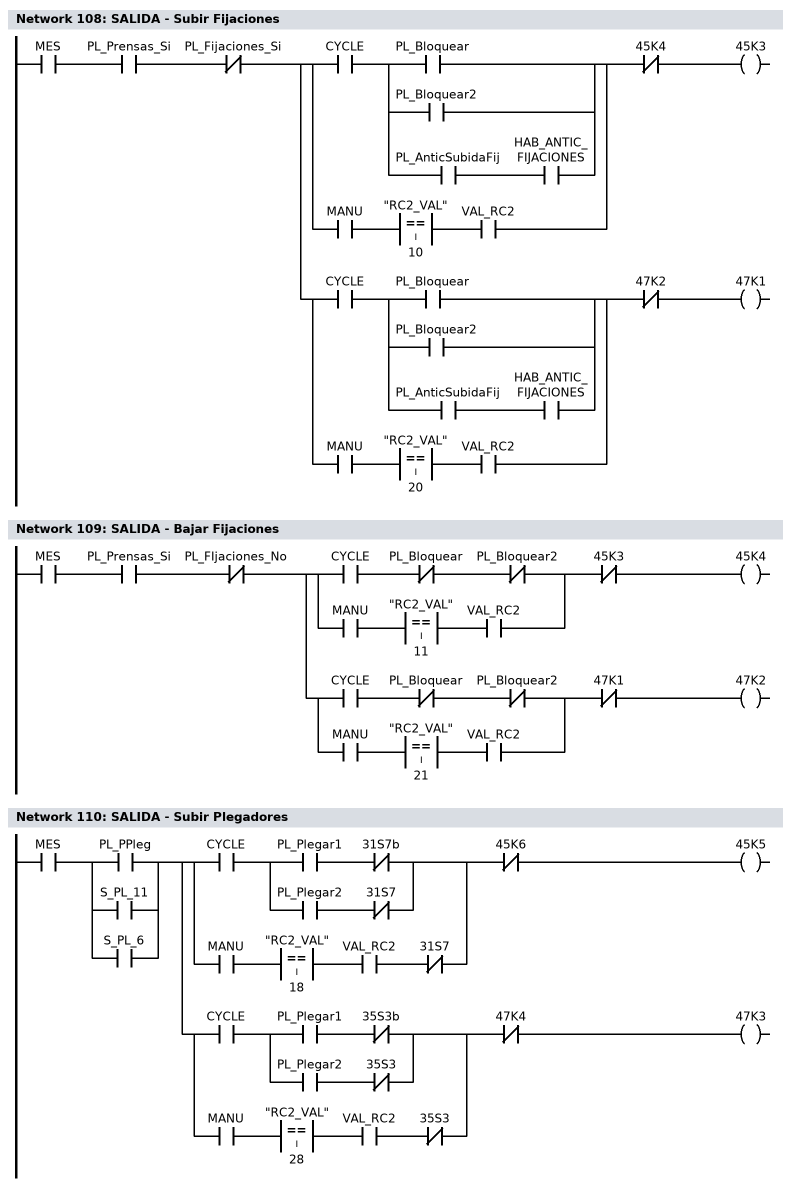
NETWORK
TITLE = SALIDA - Subir Fijaciones
      A     "MES";
      A     "PL_Prensas_Si";
      AN    "PL_Fijaciones_Si";
      =     L 98.0;
      A     L 98.0;
      A(;
      A     "CYCLE";
      A(;
      O     "PL_Bloquear";
      O     "PL_Bloquear2";
      O;
      A     "PL_AnticSubidaFij";
      A     "HAB_ANTIC_FIJACIONES";
      );
      O;
      A     "MANU";
      A(;
      L     "RC2_VAL";
      L     10;
      ==I;
      );
      A     "VAL_RC2";
      );
      AN    "45K4";
      =     "45K3";
      A     L 98.0;
      A(;
      A     "CYCLE";
      A(;
      O     "PL_Bloquear";
      O     "PL_Bloquear2";
      O;
      A     "PL_AnticSubidaFij";
      A     "HAB_ANTIC_FIJACIONES";
      );
      O;
      A     "MANU";
      A(;
      L     "RC2_VAL";
      L     20;
      ==I;
      );
      A     "VAL_RC2";
      );
      AN    "47K2";
      =     "47K1";
NETWORK
TITLE = SALIDA - Bajar Fijaciones
      A     "MES";
      A     "PL_Prensas_Si";
      AN    "PL_FIjaciones_No";
      =     L 98.0;
      A     L 98.0;
      A(;
      A     "CYCLE";
      AN    "PL_Bloquear";
      AN    "PL_Bloquear2";
      O;
      A     "MANU";
      A(;
      L     "RC2_VAL";
      L     11;
      ==I;
      );
      A     "VAL_RC2";
      );
      AN    "45K3";
      =     "45K4";
      A     L 98.0;
      A(;
      A     "CYCLE";
      AN    "PL_Bloquear";
      AN    "PL_Bloquear2";
      O;
      A     "MANU";
      A(;
      L     "RC2_VAL";
      L     21;
      ==I;
      );
      A     "VAL_RC2";
      );
      AN    "47K1";
      =     "47K2";
NETWORK
TITLE = SALIDA - Subir Plegadores
      A     "MES";
      A(;
      O     "PL_PPleg";
      O     "S_PL_11";
      O     "S_PL_6";
      );
      =     L 98.0;
      A     L 98.0;
      A(;
      A     "CYCLE";
      A(;
      A     "PL_Plegar1";
      AN    "31S7b";
      O;
      A     "PL_Plegar2";
      AN    "31S7";
      );
      O;
      A     "MANU";
      A(;
      L     "RC2_VAL";
      L     18;
      ==I;
      );
      A     "VAL_RC2";
      AN    "31S7";
      );
      AN    "45K6";
      =     "45K5";
      A     L 98.0;
      A(;
      A     "CYCLE";
      A(;
      A     "PL_Plegar1";
      AN    "35S3b";
      O;
      A     "PL_Plegar2";
      AN    "35S3";
      );
      O;
      A     "MANU";
      A(;
      L     "RC2_VAL";
      L     28;
      ==I;
      );
      A     "VAL_RC2";
      AN    "35S3";
      );
      AN    "47K4";
      =     "47K3";
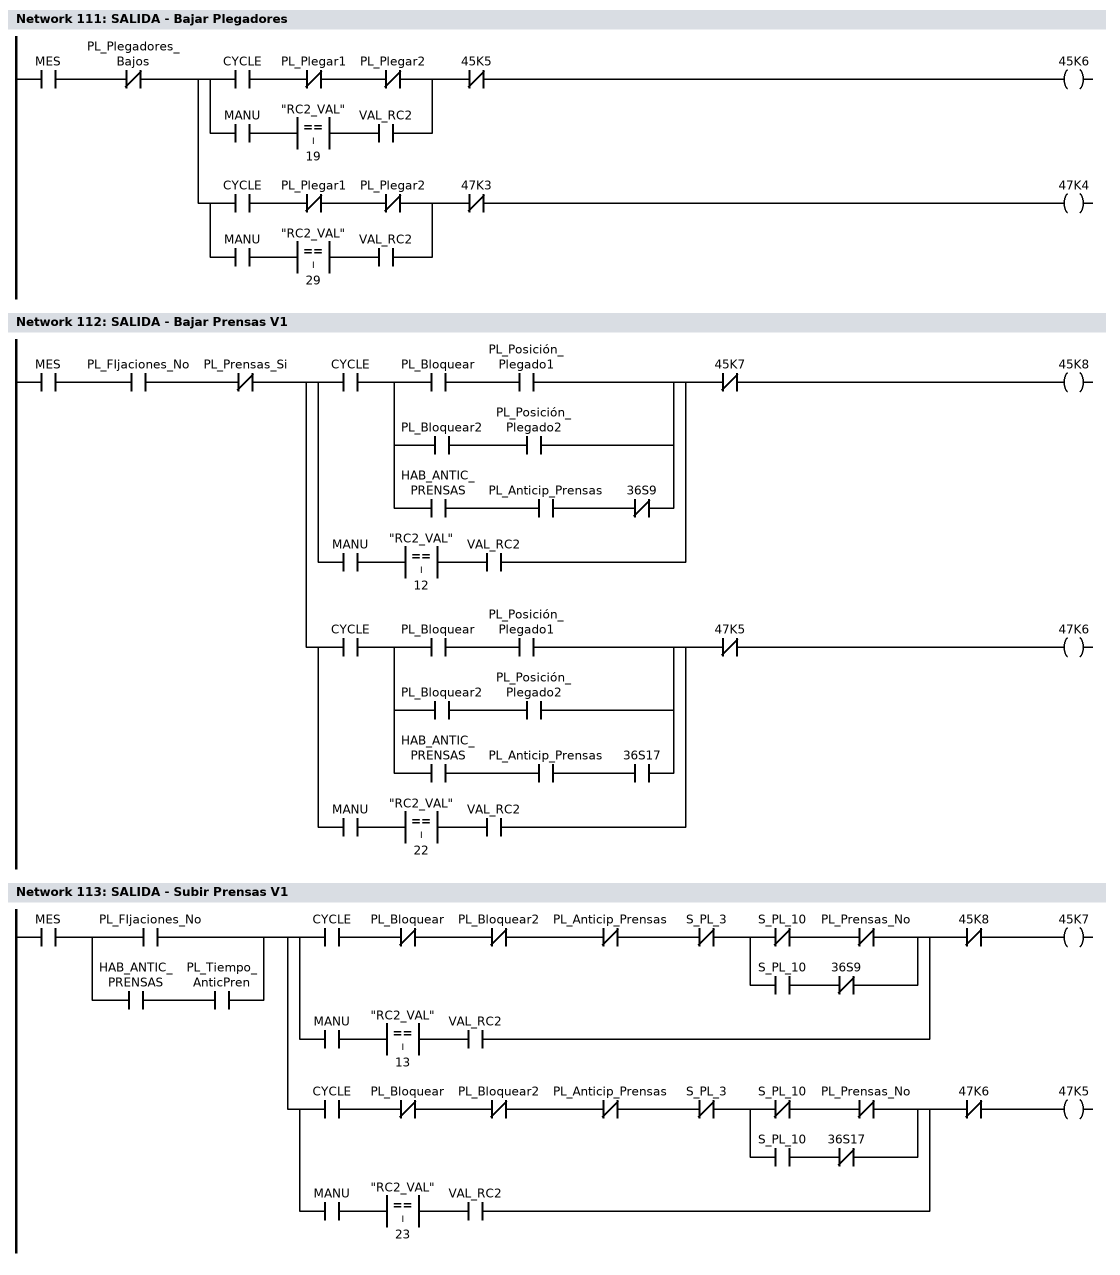
NETWORK
TITLE = SALIDA - Bajar Plegadores
      A     "MES";
      AN    "PL_Plegadores_Bajos";
      =     L 98.0;
      A     L 98.0;
      A(;
      A     "CYCLE";
      AN    "PL_Plegar1";
      AN    "PL_Plegar2";
      O;
      A     "MANU";
      A(;
      L     "RC2_VAL";
      L     19;
      ==I;
      );
      A     "VAL_RC2";
      );
      AN    "45K5";
      =     "45K6";
      A     L 98.0;
      A(;
      A     "CYCLE";
      AN    "PL_Plegar1";
      AN    "PL_Plegar2";
      O;
      A     "MANU";
      A(;
      L     "RC2_VAL";
      L     29;
      ==I;
      );
      A     "VAL_RC2";
      );
      AN    "47K3";
      =     "47K4";
NETWORK
TITLE = SALIDA - Bajar Prensas V1
      A     "MES";
      A     "PL_FIjaciones_No";
      AN    "PL_Prensas_Si";
      =     L 98.0;
      A     L 98.0;
      A(;
      A     "CYCLE";
      A(;
      A     "PL_Bloquear";
      A     "PL_Posición_Plegado1";
      O;
      A     "PL_Bloquear2";
      A     "PL_Posición_Plegado2";
      O;
      A     "HAB_ANTIC_PRENSAS";
      A     "PL_Anticip_Prensas";
      AN    "36S9";
      );
      O;
      A     "MANU";
      A(;
      L     "RC2_VAL";
      L     12;
      ==I;
      );
      A     "VAL_RC2";
      );
      AN    "45K7";
      =     "45K8";
      A     L 98.0;
      A(;
      A     "CYCLE";
      A(;
      A     "PL_Bloquear";
      A     "PL_Posición_Plegado1";
      O;
      A     "PL_Bloquear2";
      A     "PL_Posición_Plegado2";
      O;
      A     "HAB_ANTIC_PRENSAS";
      A     "PL_Anticip_Prensas";
      A     "36S17";
      );
      O;
      A     "MANU";
      A(;
      L     "RC2_VAL";
      L     22;
      ==I;
      );
      A     "VAL_RC2";
      );
      AN    "47K5";
      =     "47K6";
NETWORK
TITLE = SALIDA - Subir Prensas V1
      A     "MES";
      A(;
      O     "PL_FIjaciones_No";
      O;
      A     "HAB_ANTIC_PRENSAS";
      A     "PL_Tiempo_AnticPren";
      );
      =     L 98.0;
      A     L 98.0;
      A(;
      A     "CYCLE";
      AN    "PL_Bloquear";
      AN    "PL_Bloquear2";
      AN    "PL_Anticip_Prensas";
      AN    "S_PL_3";
      A(;
      AN    "S_PL_10";
      AN    "PL_Prensas_No";
      O;
      A     "S_PL_10";
      AN    "36S9";
      );
      O;
      A     "MANU";
      A(;
      L     "RC2_VAL";
      L     13;
      ==I;
      );
      A     "VAL_RC2";
      );
      AN    "45K8";
      =     "45K7";
      A     L 98.0;
      A(;
      A     "CYCLE";
      AN    "PL_Bloquear";
      AN    "PL_Bloquear2";
      AN    "PL_Anticip_Prensas";
      AN    "S_PL_3";
      A(;
      AN    "S_PL_10";
      AN    "PL_Prensas_No";
      O;
      A     "S_PL_10";
      AN    "36S17";
      );
      O;
      A     "MANU";
      A(;
      L     "RC2_VAL";
      L     23;
      ==I;
      );
      A     "VAL_RC2";
      );
      AN    "47K6";
      =     "47K5";
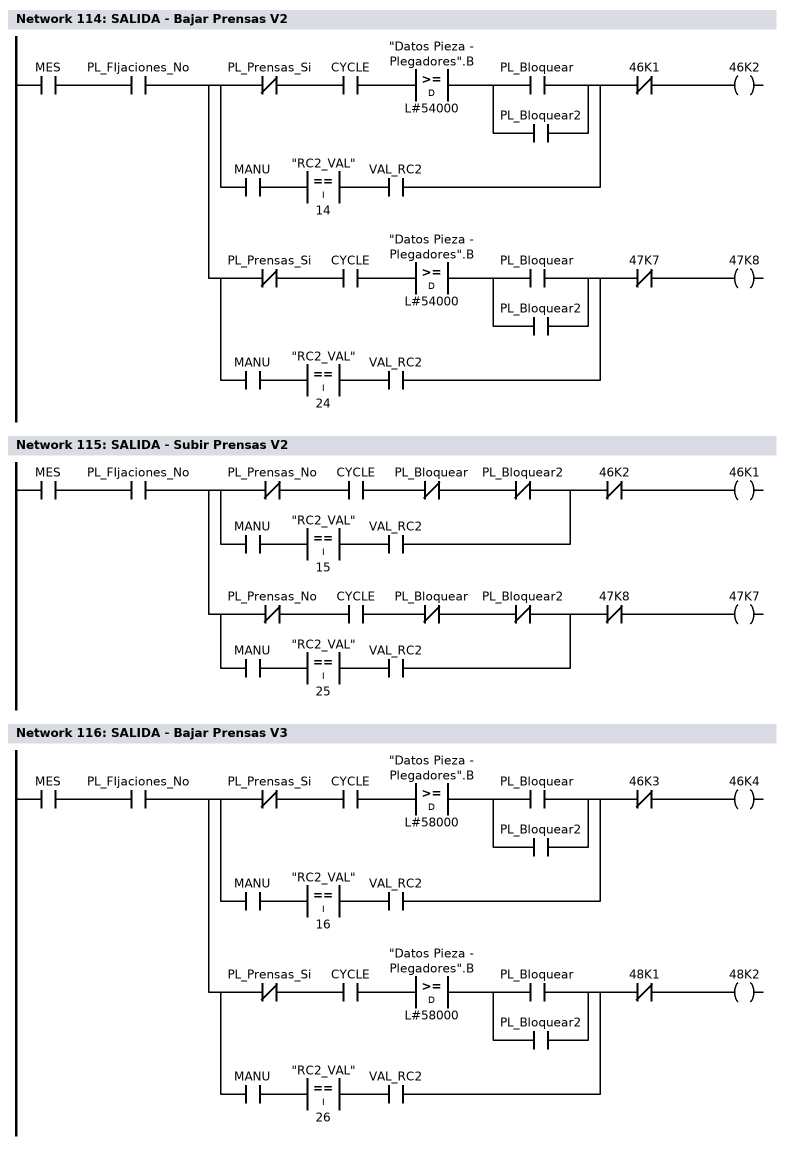
NETWORK
TITLE = SALIDA - Bajar Prensas V2
      A     "MES";
      A     "PL_FIjaciones_No";
      =     L 98.0;
      A     L 98.0;
      A(;
      AN    "PL_Prensas_Si";
      A     "CYCLE";
      A(;
      L     "Datos Pieza - Plegadores".B;
      L     L#54000;
      >=D;
      );
      A(;
      O     "PL_Bloquear";
      O     "PL_Bloquear2";
      );
      O;
      A     "MANU";
      A(;
      L     "RC2_VAL";
      L     14;
      ==I;
      );
      A     "VAL_RC2";
      );
      AN    "46K1";
      =     "46K2";
      A     L 98.0;
      A(;
      AN    "PL_Prensas_Si";
      A     "CYCLE";
      A(;
      L     "Datos Pieza - Plegadores".B;
      L     L#54000;
      >=D;
      );
      A(;
      O     "PL_Bloquear";
      O     "PL_Bloquear2";
      );
      O;
      A     "MANU";
      A(;
      L     "RC2_VAL";
      L     24;
      ==I;
      );
      A     "VAL_RC2";
      );
      AN    "47K7";
      =     "47K8";
NETWORK
TITLE = SALIDA - Subir Prensas V2
      A     "MES";
      A     "PL_FIjaciones_No";
      =     L 98.0;
      A     L 98.0;
      A(;
      AN    "PL_Prensas_No";
      A     "CYCLE";
      AN    "PL_Bloquear";
      AN    "PL_Bloquear2";
      O;
      A     "MANU";
      A(;
      L     "RC2_VAL";
      L     15;
      ==I;
      );
      A     "VAL_RC2";
      );
      AN    "46K2";
      =     "46K1";
      A     L 98.0;
      A(;
      AN    "PL_Prensas_No";
      A     "CYCLE";
      AN    "PL_Bloquear";
      AN    "PL_Bloquear2";
      O;
      A     "MANU";
      A(;
      L     "RC2_VAL";
      L     25;
      ==I;
      );
      A     "VAL_RC2";
      );
      AN    "47K8";
      =     "47K7";
NETWORK
TITLE = SALIDA - Bajar Prensas V3
      A     "MES";
      A     "PL_FIjaciones_No";
      =     L 98.0;
      A     L 98.0;
      A(;
      AN    "PL_Prensas_Si";
      A     "CYCLE";
      A(;
      L     "Datos Pieza - Plegadores".B;
      L     L#58000;
      >=D;
      );
      A(;
      O     "PL_Bloquear";
      O     "PL_Bloquear2";
      );
      O;
      A     "MANU";
      A(;
      L     "RC2_VAL";
      L     16;
      ==I;
      );
      A     "VAL_RC2";
      );
      AN    "46K3";
      =     "46K4";
      A     L 98.0;
      A(;
      AN    "PL_Prensas_Si";
      A     "CYCLE";
      A(;
      L     "Datos Pieza - Plegadores".B;
      L     L#58000;
      >=D;
      );
      A(;
      O     "PL_Bloquear";
      O     "PL_Bloquear2";
      );
      O;
      A     "MANU";
      A(;
      L     "RC2_VAL";
      L     26;
      ==I;
      );
      A     "VAL_RC2";
      );
      AN    "48K1";
      =     "48K2";
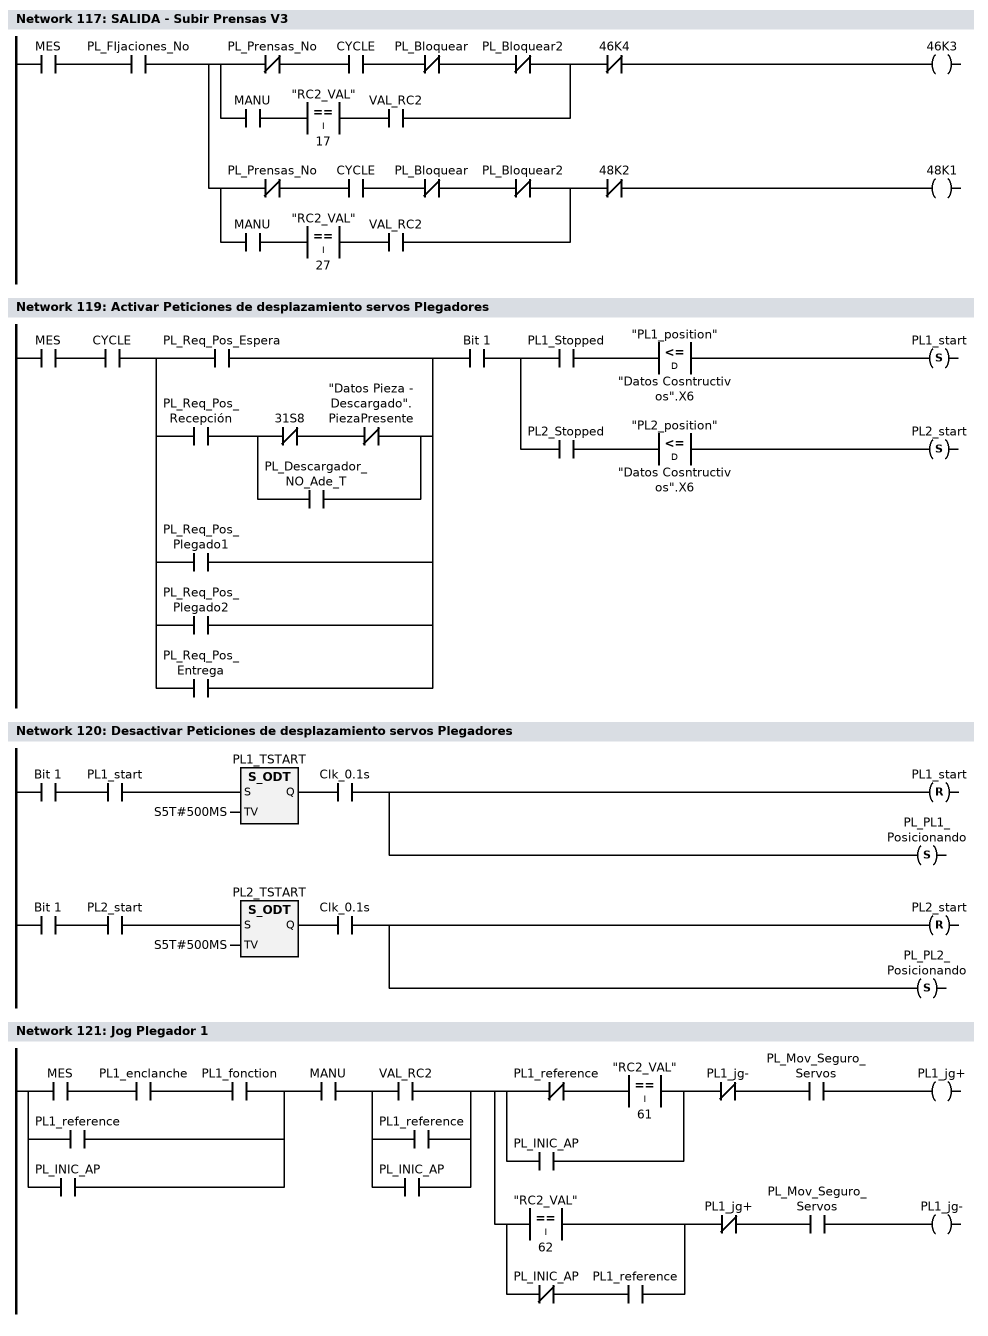
NETWORK
TITLE = SALIDA - Subir Prensas V3
      A     "MES";
      A     "PL_FIjaciones_No";
      =     L 98.0;
      A     L 98.0;
      A(;
      AN    "PL_Prensas_No";
      A     "CYCLE";
      AN    "PL_Bloquear";
      AN    "PL_Bloquear2";
      O;
      A     "MANU";
      A(;
      L     "RC2_VAL";
      L     17;
      ==I;
      );
      A     "VAL_RC2";
      );
      AN    "46K4";
      =     "46K3";
      A     L 98.0;
      A(;
      AN    "PL_Prensas_No";
      A     "CYCLE";
      AN    "PL_Bloquear";
      AN    "PL_Bloquear2";
      O;
      A     "MANU";
      A(;
      L     "RC2_VAL";
      L     27;
      ==I;
      );
      A     "VAL_RC2";
      );
      AN    "48K2";
      =     "48K1";
NETWORK
TITLE = -------------- DESPLAZAMIENTO SERVOS PLEGADORES -------------
NETWORK
TITLE = Activar Peticiones de desplazamiento servos Plegadores
      A     "MES";
      A     "CYCLE";
      A(;
      O     "PL_Req_Pos_Espera";
      O;
      A     "PL_Req_Pos_Recepción";
      A(;
      AN    "31S8";
      AN    "Datos Pieza - Descargado".PiezaPresente;
      O     "PL_Descargador_NO_Ade_T";
      );
      O     "PL_Req_Pos_Plegado1";
      O     "PL_Req_Pos_Plegado2";
      O     "PL_Req_Pos_Entrega";
      );
      A     "Bit 1";
      =     L 98.0;
      A     L 98.0;
      A     "PL1_Stopped";
      A(;
      L     "PL1_position";
      L     "Datos Cosntructivos".X6;
      <=D;
      );
      S     "PL1_start";
      A     L 98.0;
      A     "PL2_Stopped";
      A(;
      L     "PL2_position";
      L     "Datos Cosntructivos".X6;
      <=D;
      );
      S     "PL2_start";
NETWORK
TITLE = Desactivar Peticiones de desplazamiento servos Plegadores
      A     "Bit 1";
      =     L 98.0;
      A(;
      A     L 98.0;
      A     "PL1_start";
      L     S5T#500MS;
      SD    "PL1_TSTART";
      NOP   0;
      NOP   0;
      NOP   0;
      A     "PL1_TSTART";
      );
      A     "Clk_0.1s";
      R     "PL1_start";
      S     "PL_PL1_Posicionando";
      A(;
      A     L 98.0;
      A     "PL2_start";
      L     S5T#500MS;
      SD    "PL2_TSTART";
      NOP   0;
      NOP   0;
      NOP   0;
      A     "PL2_TSTART";
      );
      A     "Clk_0.1s";
      R     "PL2_start";
      S     "PL_PL2_Posicionando";
NETWORK
TITLE = Jog Plegador 1
      A(;
      A     "MES";
      A     "PL1_enclanche";
      A     "PL1_fonction";
      O     "PL1_reference";
      O     "PL_INIC_AP";
      );
      A     "MANU";
      A(;
      O     "VAL_RC2";
      O     "PL1_reference";
      O     "PL_INIC_AP";
      );
      =     L 98.0;
      A     L 98.0;
      A(;
      AN    "PL1_reference";
      A(;
      L     "RC2_VAL";
      L     61;
      ==I;
      );
      O     "PL_INIC_AP";
      );
      AN    "PL1_jg-";
      A     "PL_Mov_Seguro_Servos";
      =     "PL1_jg+";
      A     L 98.0;
      A(;
      O(;
      L     "RC2_VAL";
      L     62;
      ==I;
      );
      O;
      AN    "PL_INIC_AP";
      A     "PL1_reference";
      );
      AN    "PL1_jg+";
      A     "PL_Mov_Seguro_Servos";
      =     "PL1_jg-";
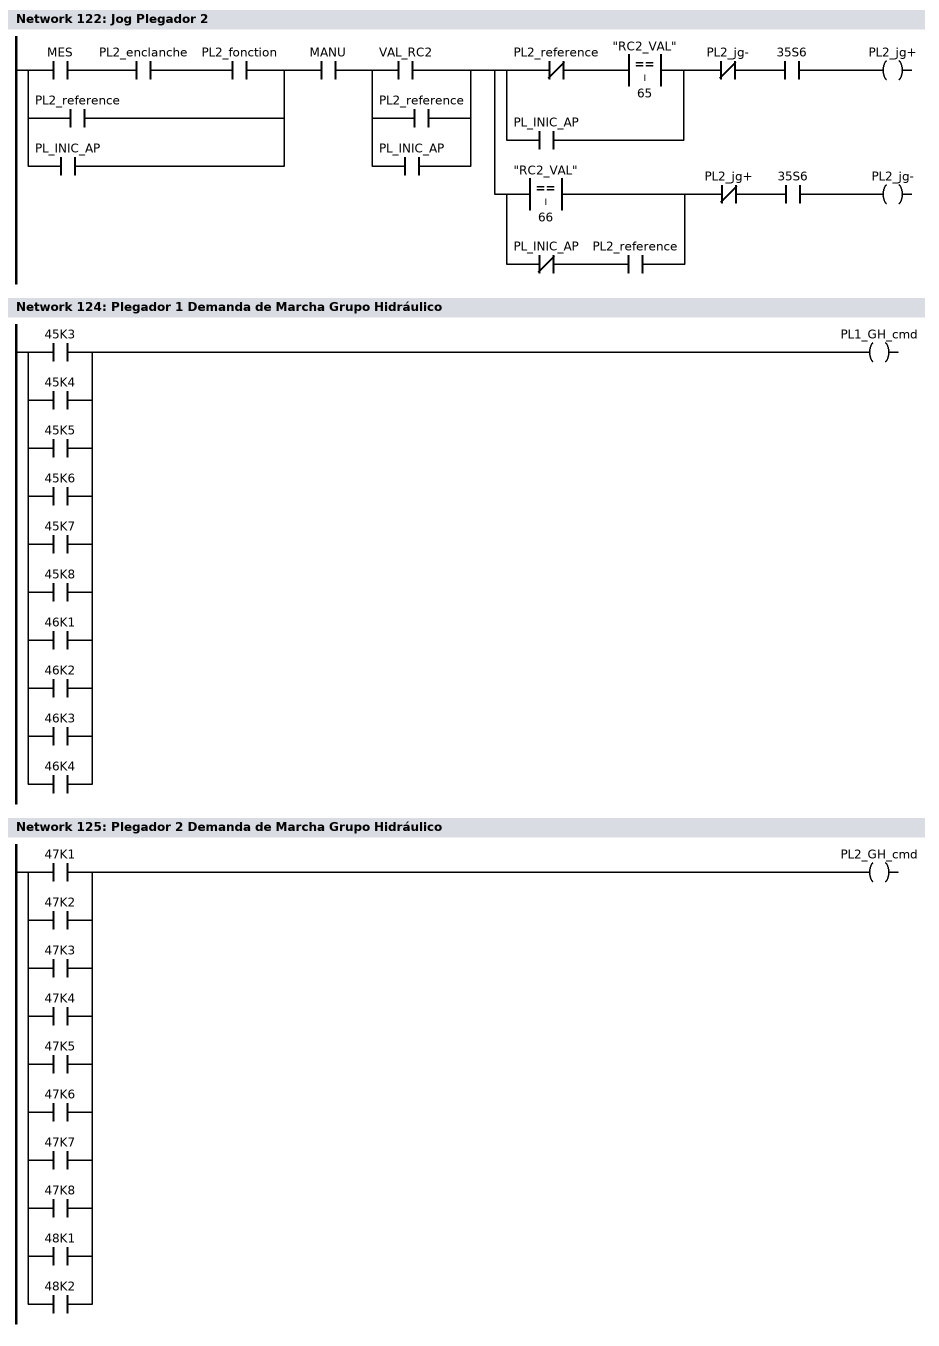
NETWORK
TITLE = Jog Plegador 2
      A(;
      A     "MES";
      A     "PL2_enclanche";
      A     "PL2_fonction";
      O     "PL2_reference";
      O     "PL_INIC_AP";
      );
      A     "MANU";
      A(;
      O     "VAL_RC2";
      O     "PL2_reference";
      O     "PL_INIC_AP";
      );
      =     L 98.0;
      A     L 98.0;
      A(;
      AN    "PL2_reference";
      A(;
      L     "RC2_VAL";
      L     65;
      ==I;
      );
      O     "PL_INIC_AP";
      );
      AN    "PL2_jg-";
      A     "35S6";
      =     "PL2_jg+";
      A     L 98.0;
      A(;
      O(;
      L     "RC2_VAL";
      L     66;
      ==I;
      );
      O;
      AN    "PL_INIC_AP";
      A     "PL2_reference";
      );
      AN    "PL2_jg+";
      A     "35S6";
      =     "PL2_jg-";
NETWORK
TITLE = --------------- CONTROL GRUPO HIDRÁULICO ------------
NETWORK
TITLE = Plegador 1 Demanda de Marcha Grupo Hidráulico
      O     "45K3";
      O     "45K4";
      O     "45K5";
      O     "45K6";
      O     "45K7";
      O     "45K8";
      O     "46K1";
      O     "46K2";
      O     "46K3";
      O     "46K4";
      =     "PL1_GH_cmd";
NETWORK
TITLE = Plegador 2 Demanda de Marcha Grupo Hidráulico
      O     "47K1";
      O     "47K2";
      O     "47K3";
      O     "47K4";
      O     "47K5";
      O     "47K6";
      O     "47K7";
      O     "47K8";
      O     "48K1";
      O     "48K2";
      =     "PL2_GH_cmd";
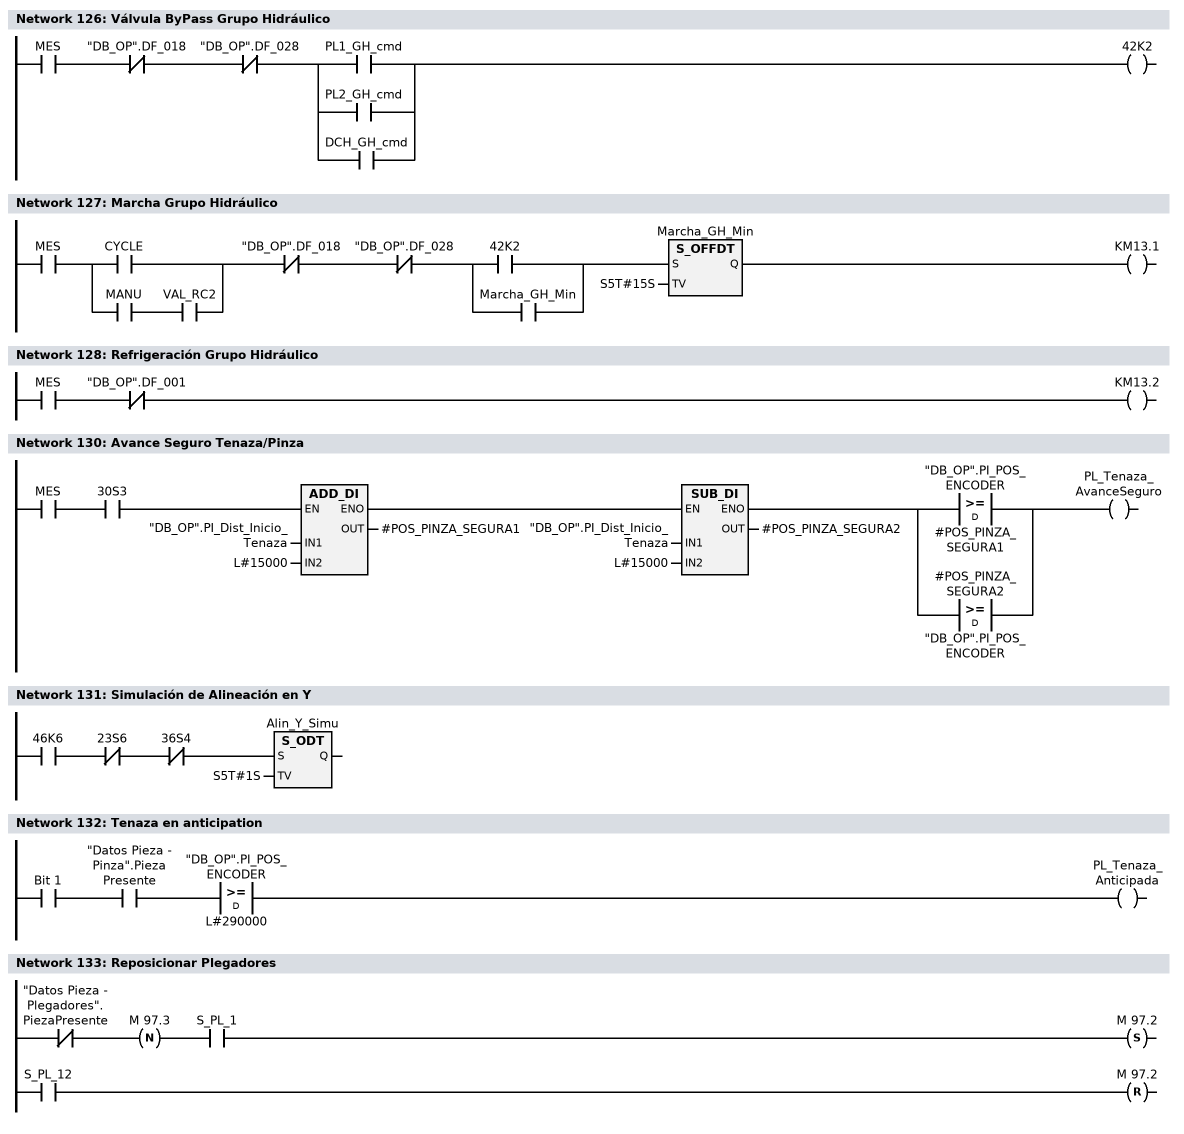
NETWORK
TITLE = Válvula ByPass Grupo Hidráulico
      A     "MES";
      AN    "DB_OP".DF_018;
      AN    "DB_OP".DF_028;
      A(;
      O     "PL1_GH_cmd";
      O     "PL2_GH_cmd";
      O     "DCH_GH_cmd";
      );
      =     "42K2";
NETWORK
TITLE = Marcha Grupo Hidráulico
      A     "MES";
      A(;
      O     "CYCLE";
      O;
      A     "MANU";
      A     "VAL_RC2";
      );
      AN    "DB_OP".DF_018;
      AN    "DB_OP".DF_028;
      A(;
      O     "42K2";
      O     "Marcha_GH_Min";
      );
      L     S5T#15S;
      SF    "Marcha_GH_Min";
      NOP   0;
      NOP   0;
      NOP   0;
      A     "Marcha_GH_Min";
      =     "KM13.1";
NETWORK
TITLE = Refrigeración Grupo Hidráulico
      A     "MES";
      AN    "DB_OP".DF_001;
      =     "KM13.2";
NETWORK
TITLE = ----------------- AUXILIARES ------------------------
NETWORK
TITLE = Avance Seguro Tenaza/Pinza
      A(;
      A(;
      A     "MES";
      A     "30S3";
      JNB   _06f;
      L     "DB_OP".PI_Dist_Inicio_Tenaza;
      L     L#15000;
      +D;
      T     #POS_PINZA_SEGURA1;
      AN    OV;
      SAVE;
      CLR;
_06f: A     BR;
      );
      JNB   _070;
      L     "DB_OP".PI_Dist_Inicio_Tenaza;
      L     L#15000;
      -D;
      T     #POS_PINZA_SEGURA2;
      AN    OV;
      SAVE;
      CLR;
_070: A     BR;
      );
      A(;
      O(;
      L     "DB_OP".PI_POS_ENCODER;
      L     #POS_PINZA_SEGURA1;
      >=D;
      );
      O(;
      L     #POS_PINZA_SEGURA2;
      L     "DB_OP".PI_POS_ENCODER;
      >=D;
      );
      );
      =     "PL_Tenaza_AvanceSeguro";
NETWORK
TITLE = Simulación de Alineación en Y
      A     "46K6";
      AN    "23S6";
      AN    "36S4";
      L     S5T#1S;
      SD    "Alin_Y_Simu";
      NOP   0;
      NOP   0;
      NOP   0;
      NOP   0;
NETWORK
TITLE = Tenaza en anticipation 
      A     "Bit 1";
      A     "Datos Pieza - Pinza".PiezaPresente;
      A(;
      L     "DB_OP".PI_POS_ENCODER;
      L     L#290000;
      >=D;
      );
      =     "PL_Tenaza_Anticipada";
NETWORK
TITLE = Reposicionar Plegadores
      AN    "Datos Pieza - Plegadores".PiezaPresente;
      FN    M 97.3;
      A     "S_PL_1";
      S     M 97.2;
      A     "S_PL_12";
      R     M 97.2;
      NOP   0;
END_FUNCTION

FUNCTION "Perfilador" : VOID	// FC 10
TITLE = Perfiladores
VERSION : 0.1
VAR_TEMP
  SECU : BOOL ;	//Seguridades
  SEL_MANU : BOOL ;	//Movimiento Manual
  NMVT : INT ;	//Numero Mouvement
  AUX_WORD : WORD ;
  AUX_REEL : REAL ;	//Auxiliar Encoder (REAL)
  AUX_DINT : DINT ;
END_VAR
BEGIN
